LIN {X 0,Y 191.848,Z 587.295,A -85,B 0,C 180,E1 -21685.798,E2 -21685.798} C_VEL
LIN {X 0,Y 192.887,Z 588.321,A -85,B 0,C 180,E1 -21690,E2 -21690} C_VEL
LIN {X 0,Y 191.871,Z 587.279,A -85,B 0,C 180,E1 -21694.201,E2 -21694.201} C_VEL
LIN {X 0,Y 191.346,Z 585.399,A -85,B 0,C 180,E1 -21697.391,E2 -21697.391} C_VEL
LIN {X 0,Y 191.276,Z 582.566,A -85,B 0,C 180,E1 -21700.586,E2 -21700.586} C_VEL
LIN {X 0,Y 191.732,Z 578.708,A -85,B 0,C 180,E1 -21703.784,E2 -21703.784} C_VEL
LIN {X 0,Y 192.838,Z 573.752,A -85,B 0,C 180,E1 -21706.951,E2 -21706.951} C_VEL
LIN {X 0,Y 194.816,Z 567.046,A -85,B 0,C 180,E1 -21710.289,E2 -21710.289} C_VEL
LIN {X 0,Y 197.119,Z 559.922,A -85,B 0,C 180,E1 -21713.09,E2 -21713.09} C_VEL
LIN {X 0,Y 199.714,Z 552.189,A -85,B 0,C 180,E1 -21715.536,E2 -21715.536} C_VEL
LIN {X 0,Y 202.715,Z 542.86,A -85,B 0,C 180,E1 -21717.906,E2 -21717.906} C_VEL
LIN {X 0,Y 205.926,Z 532.546,A -85,B 0,C 180,E1 -21719.942,E2 -21719.942} C_VEL
LIN {X 0,Y 209.011,Z 521.131,A -85,B 0,C 180,E1 -21721.694,E2 -21721.694} C_VEL
LIN {X 0,Y 211.609,Z 509.286,A -85,B 0,C 180,E1 -21723.087,E2 -21723.087} C_VEL
LIN {X 0,Y 213.648,Z 497.038,A -85,B 0,C 180,E1 -21724.145,E2 -21724.145} C_VEL
LIN {X 0,Y 215.176,Z 483.319,A -85,B 0,C 180,E1 -21724.944,E2 -21724.944} C_VEL
LIN {X 0,Y 216.382,Z 458.003,A -85,B 0,C 180,E1 -21725.811,E2 -21725.811} C_VEL
LIN {X 0,Y 214.524,Z 429.768,A -85,B 0,C 180,E1 -21727.297,E2 -21727.297} C_VEL
LIN {X 0,Y 211.874,Z 401.366,A -85,B 0,C 180,E1 -21729.012,E2 -21729.012} C_VEL
LIN {X 0,Y 211.043,Z 395.885,A -85,B 0,C 180,E1 -21729.422,E2 -21729.422} C_VEL
LIN {X 0,Y 206.302,Z 384.53,A -85,B 0,C 180,E1 -21730.977,E2 -21730.977} C_VEL
LIN {X 0,Y 200.71,Z 373.052,A -85,B 0,C 180,E1 -21732.867,E2 -21732.867} C_VEL
LIN {X 0,Y 198.537,Z 368.397,A -85,B 0,C 180,E1 -21733.75,E2 -21733.75} C_VEL
LIN {X 0,Y 196.291,Z 359.935,A -85,B 0,C 180,E1 -21737.831,E2 -21737.831} C_VEL
LIN {X 0,Y 194.026,Z 352.255,A -85,B 0,C 180,E1 -21741.992,E2 -21741.992} C_VEL
LIN {X 0,Y 192.578,Z 347.556,A -85,B 0,C 180,E1 -21744.836,E2 -21744.836} C_VEL
LIN {X 0,Y 192.567,Z 347.483,A -85,B 0,C 180,E1 -21749.273,E2 -21749.273} C_VEL
LIN {X 0,Y 192.616,Z 347.458,A -85,B 0,C 180,E1 -21751.684,E2 -21751.684} C_VEL
LIN {X 0,Y 192.669,Z 347.47,A -85,B 0,C 180,E1 -21756.344,E2 -21756.344} C_VEL
LIN {X 0,Y 192.728,Z 347.448,A -85,B 0,C 180,E1 -21761.459,E2 -21761.459} C_VEL
LIN {X 0,Y 192.755,Z 347.462,A -85,B 0,C 180,E1 -21765.213,E2 -21765.213} C_VEL
LIN {X 0,Y 192.942,Z 347.448,A -85,B 0,C 180,E1 -21769.567,E2 -21769.567} C_VEL
LIN {X 0,Y 192.965,Z 347.423,A -85,B 0,C 180,E1 -21773.727,E2 -21773.727} C_VEL
LIN {X 0,Y 193.228,Z 347.414,A -85,B 0,C 180,E1 -21777.916,E2 -21777.916} C_VEL
LIN {X 0,Y 193.409,Z 347.368,A -85,B 0,C 180,E1 -21780,E2 -21780} C_VEL
LIN {X 0,Y 192.937,Z 347.452,A -85,B 0,C 180,E1 -21784.178,E2 -21784.178} C_VEL
LIN {X 0,Y 193.02,Z 347.415,A -85,B 0,C 180,E1 -21788.375,E2 -21788.375} C_VEL
LIN {X 0,Y 192.789,Z 347.457,A -85,B 0,C 180,E1 -21792.634,E2 -21792.634} C_VEL
LIN {X 0,Y 192.716,Z 347.474,A -85,B 0,C 180,E1 -21796.963,E2 -21796.963} C_VEL
LIN {X 0,Y 192.583,Z 347.474,A -85,B 0,C 180,E1 -21801.404,E2 -21801.404} C_VEL
LIN {X 0,Y 192.624,Z 347.491,A -85,B 0,C 180,E1 -21804.199,E2 -21804.199} C_VEL
LIN {X 0,Y 192.597,Z 347.42,A -85,B 0,C 180,E1 -21808.865,E2 -21808.865} C_VEL
LIN {X 0,Y 192.592,Z 347.466,A -85,B 0,C 180,E1 -21813.187,E2 -21813.187} C_VEL
LIN {X 0,Y 192.539,Z 347.449,A -85,B 0,C 180,E1 -21818.355,E2 -21818.355} C_VEL
LIN {X 0,Y 192.504,Z 347.505,A -85,B 0,C 180,E1 -21823.101,E2 -21823.101} C_VEL
LIN {X 0,Y 192.582,Z 347.745,A -85,B 0,C 180,E1 -21825.324,E2 -21825.324} C_VEL
LIN {X 0,Y 192.845,Z 348.9,A -85,B 0,C 180,E1 -21825.748,E2 -21825.748} C_VEL
LIN {X 0,Y 194.502,Z 351.576,A -85,B 0,C 180,E1 -21826.395,E2 -21826.395} C_VEL
LIN {X 0,Y 195.588,Z 352.693,A -85,B 0,C 180,E1 -21826.764,E2 -21826.764} C_VEL
LIN {X 0,Y 197.832,Z 356.164,A -85,B 0,C 180,E1 -21827.564,E2 -21827.564} C_VEL
LIN {X 0,Y 203.879,Z 365.281,A -85,B 0,C 180,E1 -21829.573,E2 -21829.573} C_VEL
LIN {X 0,Y 210.142,Z 375.738,A -85,B 0,C 180,E1 -21831.518,E2 -21831.518} C_VEL
LIN {X 0,Y 216.801,Z 388.352,A -85,B 0,C 180,E1 -21833.471,E2 -21833.471} C_VEL
LIN {X 0,Y 219.395,Z 393.771,A -85,B 0,C 180,E1 -21834.207,E2 -21834.207} C_VEL
LIN {X 0,Y 218.184,Z 433.029,A -85,B 0,C 180,E1 -21835.609,E2 -21835.609} C_VEL
LIN {X 0,Y 217.164,Z 446.771,A -85,B 0,C 180,E1 -21836.484,E2 -21836.484} C_VEL
LIN {X 0,Y 215.726,Z 459.041,A -85,B 0,C 180,E1 -21837.637,E2 -21837.637} C_VEL
LIN {X 0,Y 213.801,Z 470.392,A -85,B 0,C 180,E1 -21839.058,E2 -21839.058} C_VEL
LIN {X 0,Y 211.456,Z 480.568,A -85,B 0,C 180,E1 -21840.645,E2 -21840.645} C_VEL
LIN {X 0,Y 209.005,Z 489.845,A -85,B 0,C 180,E1 -21842.461,E2 -21842.461} C_VEL
LIN {X 0,Y 206.379,Z 499.292,A -85,B 0,C 180,E1 -21844.807,E2 -21844.807} C_VEL
LIN {X 0,Y 203.892,Z 507.03,A -85,B 0,C 180,E1 -21847.184,E2 -21847.184} C_VEL
LIN {X 0,Y 201.23,Z 514.686,A -85,B 0,C 180,E1 -21850.145,E2 -21850.145} C_VEL
LIN {X 0,Y 198.708,Z 521.487,A -85,B 0,C 180,E1 -21853.564,E2 -21853.564} C_VEL
LIN {X 0,Y 196.834,Z 526.095,A -85,B 0,C 180,E1 -21856.58,E2 -21856.58} C_VEL
LIN {X 0,Y 195.194,Z 529.639,A -85,B 0,C 180,E1 -21859.629,E2 -21859.629} C_VEL
LIN {X 0,Y 194.393,Z 531.461,A -85,B 0,C 180,E1 -21861.685,E2 -21861.685} C_VEL
LIN {X 0,Y 194.029,Z 532.795,A -85,B 0,C 180,E1 -21863.762,E2 -21863.762} C_VEL
LIN {X 0,Y 193.592,Z 533.767,A -85,B 0,C 180,E1 -21865.836,E2 -21865.836} C_VEL
LIN {X 0,Y 193.485,Z 534.343,A -85,B 0,C 180,E1 -21867.918,E2 -21867.918} C_VEL
LIN {X 0,Y 193.415,Z 534.565,A -85,B 0,C 180,E1 -21870,E2 -21870} C_VEL
LIN {X 0,Y 193.484,Z 534.376,A -85,B 0,C 180,E1 -21872.082,E2 -21872.082} C_VEL
LIN {X 0,Y 194.022,Z 532.87,A -85,B 0,C 180,E1 -21876.238,E2 -21876.238} C_VEL
LIN {X 0,Y 194.377,Z 531.572,A -85,B 0,C 180,E1 -21878.316,E2 -21878.316} C_VEL
LIN {X 0,Y 195.772,Z 528.732,A -85,B 0,C 180,E1 -21881.387,E2 -21881.387} C_VEL
LIN {X 0,Y 197.474,Z 524.899,A -85,B 0,C 180,E1 -21884.426,E2 -21884.426} C_VEL
LIN {X 0,Y 199.366,Z 519.811,A -85,B 0,C 180,E1 -21887.541,E2 -21887.541} C_VEL
LIN {X 0,Y 202.139,Z 512.562,A -85,B 0,C 180,E1 -21890.877,E2 -21890.877} C_VEL
LIN {X 0,Y 204.908,Z 504.527,A -85,B 0,C 180,E1 -21893.766,E2 -21893.766} C_VEL
LIN {X 0,Y 207.391,Z 496.296,A -85,B 0,C 180,E1 -21896.138,E2 -21896.138} C_VEL
LIN {X 0,Y 209.819,Z 487.254,A -85,B 0,C 180,E1 -21898.237,E2 -21898.237} C_VEL
LIN {X 0,Y 212.577,Z 476.707,A -85,B 0,C 180,E1 -21900.126,E2 -21900.126} C_VEL
LIN {X 0,Y 214.853,Z 465.168,A -85,B 0,C 180,E1 -21901.781,E2 -21901.781} C_VEL
LIN {X 0,Y 216.678,Z 453.863,A -85,B 0,C 180,E1 -21903.004,E2 -21903.004} C_VEL
LIN {X 0,Y 217.809,Z 441.291,A -85,B 0,C 180,E1 -21904.043,E2 -21904.043} C_VEL
LIN {X 0,Y 218.404,Z 428.456,A -85,B 0,C 180,E1 -21904.744,E2 -21904.744} C_VEL
LIN {X 0,Y 219.541,Z 393.957,A -85,B 0,C 180,E1 -21905.916,E2 -21905.916} C_VEL
LIN {X 0,Y 211.91,Z 378.784,A -85,B 0,C 180,E1 -21908.126,E2 -21908.126} C_VEL
LIN {X 0,Y 205.192,Z 367.34,A -85,B 0,C 180,E1 -21910.185,E2 -21910.185} C_VEL
LIN {X 0,Y 198.147,Z 356.536,A -85,B 0,C 180,E1 -21912.516,E2 -21912.516} C_VEL
LIN {X 0,Y 195.883,Z 353.302,A -85,B 0,C 180,E1 -21913.309,E2 -21913.309} C_VEL
LIN {X 0,Y 194.98,Z 352.019,A -85,B 0,C 180,E1 -21913.633,E2 -21913.633} C_VEL
LIN {X 0,Y 193.09,Z 349.489,A -85,B 0,C 180,E1 -21914.325,E2 -21914.325} C_VEL
LIN {X 0,Y 192.625,Z 347.931,A -85,B 0,C 180,E1 -21914.751,E2 -21914.751} C_VEL
LIN {X 0,Y 192.543,Z 347.583,A -85,B 0,C 180,E1 -21915.101,E2 -21915.101} C_VEL
LIN {X 0,Y 192.503,Z 347.454,A -85,B 0,C 180,E1 -21920.055,E2 -21920.055} C_VEL
LIN {X 0,Y 192.556,Z 347.486,A -85,B 0,C 180,E1 -21924.269,E2 -21924.269} C_VEL
LIN {X 0,Y 192.603,Z 347.46,A -85,B 0,C 180,E1 -21927.061,E2 -21927.061} C_VEL
LIN {X 0,Y 192.616,Z 347.421,A -85,B 0,C 180,E1 -21931.684,E2 -21931.684} C_VEL
LIN {X 0,Y 192.659,Z 347.486,A -85,B 0,C 180,E1 -21936.342,E2 -21936.342} C_VEL
LIN {X 0,Y 192.692,Z 347.48,A -85,B 0,C 180,E1 -21941.491,E2 -21941.491} C_VEL
LIN {X 0,Y 192.725,Z 347.453,A -85,B 0,C 180,E1 -21945.211,E2 -21945.211} C_VEL
LIN {X 0,Y 192.943,Z 347.447,A -85,B 0,C 180,E1 -21949.567,E2 -21949.567} C_VEL
LIN {X 0,Y 192.962,Z 347.432,A -85,B 0,C 180,E1 -21953.727,E2 -21953.727} C_VEL
LIN {X 0,Y 193.228,Z 347.394,A -85,B 0,C 180,E1 -21957.915,E2 -21957.915} C_VEL
LIN {X 0,Y 193.409,Z 347.368,A -85,B 0,C 180,E1 -21960,E2 -21960} C_VEL
LIN {X 0,Y 192.932,Z 347.439,A -85,B 0,C 180,E1 -21964.178,E2 -21964.178} C_VEL
LIN {X 0,Y 193.021,Z 347.433,A -85,B 0,C 180,E1 -21968.374,E2 -21968.374} C_VEL
LIN {X 0,Y 192.79,Z 347.445,A -85,B 0,C 180,E1 -21972.634,E2 -21972.634} C_VEL
LIN {X 0,Y 192.743,Z 347.472,A -85,B 0,C 180,E1 -21976.96,E2 -21976.96} C_VEL
LIN {X 0,Y 192.589,Z 347.45,A -85,B 0,C 180,E1 -21981.403,E2 -21981.403} C_VEL
LIN {X 0,Y 192.632,Z 347.487,A -85,B 0,C 180,E1 -21984.205,E2 -21984.205} C_VEL
LIN {X 0,Y 192.598,Z 347.461,A -85,B 0,C 180,E1 -21988.865,E2 -21988.865} C_VEL
LIN {X 0,Y 192.592,Z 347.477,A -85,B 0,C 180,E1 -21993.187,E2 -21993.187} C_VEL
LIN {X 0,Y 192.586,Z 347.766,A -85,B 0,C 180,E1 -21995.243,E2 -21995.243} C_VEL
LIN {X 0,Y 195.04,Z 355.553,A -85,B 0,C 180,E1 -21999.762,E2 -21999.762} C_VEL
LIN {X 0,Y 197.364,Z 363.876,A -85,B 0,C 180,E1 -22004.064,E2 -22004.064} C_VEL
LIN {X 0,Y 198.612,Z 368.614,A -85,B 0,C 180,E1 -22006.227,E2 -22006.227} C_VEL
LIN {X 0,Y 204.695,Z 381.021,A -85,B 0,C 180,E1 -22008.404,E2 -22008.404} C_VEL
LIN {X 0,Y 210.896,Z 395.328,A -85,B 0,C 180,E1 -22010.448,E2 -22010.448} C_VEL
LIN {X 0,Y 211.406,Z 397.261,A -85,B 0,C 180,E1 -22010.64,E2 -22010.64} C_VEL
LIN {X 0,Y 213.526,Z 416.852,A -85,B 0,C 180,E1 -22011.904,E2 -22011.904} C_VEL
LIN {X 0,Y 216.009,Z 448.818,A -85,B 0,C 180,E1 -22013.687,E2 -22013.687} C_VEL
LIN {X 0,Y 216.547,Z 458.703,A -85,B 0,C 180,E1 -22014.181,E2 -22014.181} C_VEL
LIN {X 0,Y 215.968,Z 464.541,A -85,B 0,C 180,E1 -22014.299,E2 -22014.299} C_VEL
LIN {X 0,Y 213.192,Z 474.039,A -85,B 0,C 180,E1 -22014.169,E2 -22014.169} C_VEL
LIN {X 0,Y 210.01,Z 483.484,A -85,B 0,C 180,E1 -22014.056,E2 -22014.056} C_VEL
LIN {X 0,Y 208.832,Z 489.253,A -85,B 0,C 180,E1 -22014.263,E2 -22014.263} C_VEL
LIN {X 0,Y 207.17,Z 500.744,A -85,B 0,C 180,E1 -22015.078,E2 -22015.078} C_VEL
LIN {X 0,Y 205.007,Z 511.757,A -85,B 0,C 180,E1 -22016.147,E2 -22016.147} C_VEL
LIN {X 0,Y 202.148,Z 523.63,A -85,B 0,C 180,E1 -22017.688,E2 -22017.688} C_VEL
LIN {X 0,Y 198.624,Z 535.483,A -85,B 0,C 180,E1 -22019.721,E2 -22019.721} C_VEL
LIN {X 0,Y 195.149,Z 546.05,A -85,B 0,C 180,E1 -22022.085,E2 -22022.085} C_VEL
LIN {X 0,Y 192.136,Z 554.643,A -85,B 0,C 180,E1 -22024.546,E2 -22024.546} C_VEL
LIN {X 0,Y 189.191,Z 563.086,A -85,B 0,C 180,E1 -22027.619,E2 -22027.619} C_VEL
LIN {X 0,Y 186.75,Z 569.919,A -85,B 0,C 180,E1 -22030.775,E2 -22030.775} C_VEL
LIN {X 0,Y 185.118,Z 576.286,A -85,B 0,C 180,E1 -22034.588,E2 -22034.588} C_VEL
LIN {X 0,Y 184.32,Z 580.472,A -85,B 0,C 180,E1 -22037.895,E2 -22037.895} C_VEL
LIN {X 0,Y 184.177,Z 583.631,A -85,B 0,C 180,E1 -22041.22,E2 -22041.22} C_VEL
LIN {X 0,Y 184.38,Z 585.174,A -85,B 0,C 180,E1 -22043.434,E2 -22043.434} C_VEL
LIN {X 0,Y 184.755,Z 586.306,A -85,B 0,C 180,E1 -22045.637,E2 -22045.637} C_VEL
LIN {X 0,Y 185.837,Z 587.34,A -85,B 0,C 180,E1 -22050,E2 -22050} C_VEL
LIN {X 0,Y 184.774,Z 586.288,A -85,B 0,C 180,E1 -22054.363,E2 -22054.363} C_VEL
LIN {X 0,Y 184.289,Z 584.561,A -85,B 0,C 180,E1 -22057.461,E2 -22057.461} C_VEL
LIN {X 0,Y 184.232,Z 581.567,A -85,B 0,C 180,E1 -22060.996,E2 -22060.996} C_VEL
LIN {X 0,Y 184.764,Z 577.708,A -85,B 0,C 180,E1 -22064.314,E2 -22064.314} C_VEL
LIN {X 0,Y 185.968,Z 572.749,A -85,B 0,C 180,E1 -22067.597,E2 -22067.597} C_VEL
LIN {X 0,Y 187.904,Z 566.664,A -85,B 0,C 180,E1 -22070.763,E2 -22070.763} C_VEL
LIN {X 0,Y 190.556,Z 558.924,A -85,B 0,C 180,E1 -22073.934,E2 -22073.934} C_VEL
LIN {X 0,Y 193.301,Z 551.194,A -85,B 0,C 180,E1 -22076.447,E2 -22076.447} C_VEL
LIN {X 0,Y 196.459,Z 541.868,A -85,B 0,C 180,E1 -22078.877,E2 -22078.877} C_VEL
LIN {X 0,Y 199.812,Z 531.555,A -85,B 0,C 180,E1 -22080.957,E2 -22080.957} C_VEL
LIN {X 0,Y 203.013,Z 520.14,A -85,B 0,C 180,E1 -22082.745,E2 -22082.745} C_VEL
LIN {X 0,Y 205.657,Z 508.286,A -85,B 0,C 180,E1 -22084.174,E2 -22084.174} C_VEL
LIN {X 0,Y 207.798,Z 496.149,A -85,B 0,C 180,E1 -22085.236,E2 -22085.236} C_VEL
LIN {X 0,Y 209.337,Z 482.771,A -85,B 0,C 180,E1 -22086.039,E2 -22086.039} C_VEL
LIN {X 0,Y 210.605,Z 459.13,A -85,B 0,C 180,E1 -22086.864,E2 -22086.864} C_VEL
LIN {X 0,Y 208.769,Z 429.728,A -85,B 0,C 180,E1 -22088.468,E2 -22088.468} C_VEL
LIN {X 0,Y 205.982,Z 399.581,A -85,B 0,C 180,E1 -22090.383,E2 -22090.383} C_VEL
LIN {X 0,Y 202.843,Z 391.689,A -85,B 0,C 180,E1 -22091.474,E2 -22091.474} C_VEL
LIN {X 0,Y 196.692,Z 378.218,A -85,B 0,C 180,E1 -22093.673,E2 -22093.673} C_VEL
LIN {X 0,Y 193.129,Z 371.46,A -85,B 0,C 180,E1 -22094.996,E2 -22094.996} C_VEL
LIN {X 0,Y 190.941,Z 366.871,A -85,B 0,C 180,E1 -22095.994,E2 -22095.994} C_VEL
LIN {X 0,Y 188.512,Z 358.02,A -85,B 0,C 180,E1 -22100.67,E2 -22100.67} C_VEL
LIN {X 0,Y 186.002,Z 350.11,A -85,B 0,C 180,E1 -22105.475,E2 -22105.475} C_VEL
LIN {X 0,Y 185.573,Z 348.398,A -85,B 0,C 180,E1 -22106.64,E2 -22106.64} C_VEL
LIN {X 0,Y 185.544,Z 348.342,A -85,B 0,C 180,E1 -22110.595,E2 -22110.595} C_VEL
LIN {X 0,Y 185.578,Z 348.369,A -85,B 0,C 180,E1 -22115.381,E2 -22115.381} C_VEL
LIN {X 0,Y 185.67,Z 348.321,A -85,B 0,C 180,E1 -22121.135,E2 -22121.135} C_VEL
LIN {X 0,Y 185.687,Z 348.35,A -85,B 0,C 180,E1 -22124.637,E2 -22124.637} C_VEL
LIN {X 0,Y 185.885,Z 348.325,A -85,B 0,C 180,E1 -22129.419,E2 -22129.419} C_VEL
LIN {X 0,Y 185.93,Z 348.299,A -85,B 0,C 180,E1 -22133.489,E2 -22133.489} C_VEL
LIN {X 0,Y 186.173,Z 348.293,A -85,B 0,C 180,E1 -22137.837,E2 -22137.837} C_VEL
LIN {X 0,Y 186.375,Z 348.244,A -85,B 0,C 180,E1 -22140,E2 -22140} C_VEL
LIN {X 0,Y 185.885,Z 348.33,A -85,B 0,C 180,E1 -22144.337,E2 -22144.337} C_VEL
LIN {X 0,Y 185.97,Z 348.295,A -85,B 0,C 180,E1 -22148.695,E2 -22148.695} C_VEL
LIN {X 0,Y 185.714,Z 348.332,A -85,B 0,C 180,E1 -22153.124,E2 -22153.124} C_VEL
LIN {X 0,Y 185.653,Z 348.359,A -85,B 0,C 180,E1 -22157.629,E2 -22157.629} C_VEL
LIN {X 0,Y 185.55,Z 348.355,A -85,B 0,C 180,E1 -22162.257,E2 -22162.257} C_VEL
LIN {X 0,Y 185.497,Z 348.324,A -85,B 0,C 180,E1 -22167.043,E2 -22167.043} C_VEL
LIN {X 0,Y 185.541,Z 348.296,A -85,B 0,C 180,E1 -22169.5,E2 -22169.5} C_VEL
LIN {X 0,Y 185.495,Z 348.38,A -85,B 0,C 180,E1 -22174.633,E2 -22174.633} C_VEL
LIN {X 0,Y 185.498,Z 348.335,A -85,B 0,C 180,E1 -22177.315,E2 -22177.315} C_VEL
LIN {X 0,Y 185.49,Z 348.481,A -85,B 0,C 180,E1 -22182.922,E2 -22182.922} C_VEL
LIN {X 0,Y 185.708,Z 349.527,A -85,B 0,C 180,E1 -22183.499,E2 -22183.499} C_VEL
LIN {X 0,Y 187.062,Z 352.077,A -85,B 0,C 180,E1 -22184.129,E2 -22184.129} C_VEL
LIN {X 0,Y 188.825,Z 353.884,A -85,B 0,C 180,E1 -22184.794,E2 -22184.794} C_VEL
LIN {X 0,Y 191.08,Z 357.305,A -85,B 0,C 180,E1 -22185.675,E2 -22185.675} C_VEL
LIN {X 0,Y 195.742,Z 364.087,A -85,B 0,C 180,E1 -22187.376,E2 -22187.376} C_VEL
LIN {X 0,Y 202.922,Z 375.487,A -85,B 0,C 180,E1 -22189.806,E2 -22189.806} C_VEL
LIN {X 0,Y 209.873,Z 388.222,A -85,B 0,C 180,E1 -22191.998,E2 -22191.998} C_VEL
LIN {X 0,Y 213.666,Z 396.039,A -85,B 0,C 180,E1 -22193.144,E2 -22193.144} C_VEL
LIN {X 0,Y 212.389,Z 434.304,A -85,B 0,C 180,E1 -22194.549,E2 -22194.549} C_VEL
LIN {X 0,Y 211.33,Z 447.834,A -85,B 0,C 180,E1 -22195.437,E2 -22195.437} C_VEL
LIN {X 0,Y 209.822,Z 460.026,A -85,B 0,C 180,E1 -22196.61,E2 -22196.61} C_VEL
LIN {X 0,Y 207.841,Z 471.183,A -85,B 0,C 180,E1 -22198.032,E2 -22198.032} C_VEL
LIN {X 0,Y 205.359,Z 481.55,A -85,B 0,C 180,E1 -22199.683,E2 -22199.683} C_VEL
LIN {X 0,Y 202.797,Z 490.827,A -85,B 0,C 180,E1 -22201.543,E2 -22201.543} C_VEL
LIN {X 0,Y 200.041,Z 500.273,A -85,B 0,C 180,E1 -22203.95,E2 -22203.95} C_VEL
LIN {X 0,Y 197.433,Z 508.01,A -85,B 0,C 180,E1 -22206.393,E2 -22206.393} C_VEL
LIN {X 0,Y 194.634,Z 515.666,A -85,B 0,C 180,E1 -22209.442,E2 -22209.442} C_VEL
LIN {X 0,Y 191.978,Z 522.466,A -85,B 0,C 180,E1 -22212.971,E2 -22212.971} C_VEL
LIN {X 0,Y 190.005,Z 527.074,A -85,B 0,C 180,E1 -22216.089,E2 -22216.089} C_VEL
LIN {X 0,Y 188.282,Z 530.618,A -85,B 0,C 180,E1 -22219.244,E2 -22219.244} C_VEL
LIN {X 0,Y 187.438,Z 532.441,A -85,B 0,C 180,E1 -22221.374,E2 -22221.374} C_VEL
LIN {X 0,Y 187.042,Z 533.773,A -85,B 0,C 180,E1 -22223.528,E2 -22223.528} C_VEL
LIN {X 0,Y 186.583,Z 534.745,A -85,B 0,C 180,E1 -22225.68,E2 -22225.68} C_VEL
LIN {X 0,Y 186.462,Z 535.321,A -85,B 0,C 180,E1 -22227.84,E2 -22227.84} C_VEL
LIN {X 0,Y 186.388,Z 535.543,A -85,B 0,C 180,E1 -22230,E2 -22230} C_VEL
LIN {X 0,Y 186.461,Z 535.354,A -85,B 0,C 180,E1 -22232.16,E2 -22232.16} C_VEL
LIN {X 0,Y 187.035,Z 533.848,A -85,B 0,C 180,E1 -22236.472,E2 -22236.472} C_VEL
LIN {X 0,Y 187.421,Z 532.55,A -85,B 0,C 180,E1 -22238.626,E2 -22238.626} C_VEL
LIN {X 0,Y 188.888,Z 529.71,A -85,B 0,C 180,E1 -22241.808,E2 -22241.808} C_VEL
LIN {X 0,Y 190.676,Z 525.876,A -85,B 0,C 180,E1 -22244.952,E2 -22244.952} C_VEL
LIN {X 0,Y 192.676,Z 520.788,A -85,B 0,C 180,E1 -22248.171,E2 -22248.171} C_VEL
LIN {X 0,Y 195.588,Z 513.538,A -85,B 0,C 180,E1 -22251.611,E2 -22251.611} C_VEL
LIN {X 0,Y 198.496,Z 505.503,A -85,B 0,C 180,E1 -22254.583,E2 -22254.583} C_VEL
LIN {X 0,Y 201.103,Z 497.272,A -85,B 0,C 180,E1 -22257.02,E2 -22257.02} C_VEL
LIN {X 0,Y 203.66,Z 488.227,A -85,B 0,C 180,E1 -22259.171,E2 -22259.171} C_VEL
LIN {X 0,Y 206.799,Z 476.655,A -85,B 0,C 180,E1 -22261.266,E2 -22261.266} C_VEL
LIN {X 0,Y 209.196,Z 464.702,A -85,B 0,C 180,E1 -22262.978,E2 -22262.978} C_VEL
LIN {X 0,Y 211.103,Z 452.077,A -85,B 0,C 180,E1 -22264.309,E2 -22264.309} C_VEL
LIN {X 0,Y 212.274,Z 439.226,A -85,B 0,C 180,E1 -22265.301,E2 -22265.301} C_VEL
LIN {X 0,Y 212.795,Z 425.544,A -85,B 0,C 180,E1 -22265.973,E2 -22265.973} C_VEL
LIN {X 0,Y 213.782,Z 396.205,A -85,B 0,C 180,E1 -22266.989,E2 -22266.989} C_VEL
LIN {X 0,Y 206.699,Z 382.077,A -85,B 0,C 180,E1 -22269.162,E2 -22269.162} C_VEL
LIN {X 0,Y 200.469,Z 371.475,A -85,B 0,C 180,E1 -22271.179,E2 -22271.179} C_VEL
LIN {X 0,Y 194.162,Z 361.696,A -85,B 0,C 180,E1 -22273.379,E2 -22273.379} C_VEL
LIN {X 0,Y 191.048,Z 357.25,A -85,B 0,C 180,E1 -22274.532,E2 -22274.532} C_VEL
LIN {X 0,Y 188.907,Z 354.019,A -85,B 0,C 180,E1 -22275.37,E2 -22275.37} C_VEL
LIN {X 0,Y 186.163,Z 350.725,A -85,B 0,C 180,E1 -22276.446,E2 -22276.446} C_VEL
LIN {X 0,Y 185.603,Z 349.075,A -85,B 0,C 180,E1 -22276.845,E2 -22276.845} C_VEL
LIN {X 0,Y 185.444,Z 348.432,A -85,B 0,C 180,E1 -22277.457,E2 -22277.457} C_VEL
LIN {X 0,Y 185.499,Z 348.334,A -85,B 0,C 180,E1 -22282.713,E2 -22282.713} C_VEL
LIN {X 0,Y 185.528,Z 348.319,A -85,B 0,C 180,E1 -22287.972,E2 -22287.972} C_VEL
LIN {X 0,Y 185.545,Z 348.296,A -85,B 0,C 180,E1 -22290.595,E2 -22290.595} C_VEL
LIN {X 0,Y 185.56,Z 348.368,A -85,B 0,C 180,E1 -22295.378,E2 -22295.378} C_VEL
LIN {X 0,Y 185.622,Z 348.356,A -85,B 0,C 180,E1 -22301.178,E2 -22301.178} C_VEL
LIN {X 0,Y 185.656,Z 348.335,A -85,B 0,C 180,E1 -22304.634,E2 -22304.634} C_VEL
LIN {X 0,Y 185.885,Z 348.327,A -85,B 0,C 180,E1 -22309.419,E2 -22309.419} C_VEL
LIN {X 0,Y 185.927,Z 348.305,A -85,B 0,C 180,E1 -22313.489,E2 -22313.489} C_VEL
LIN {X 0,Y 186.174,Z 348.273,A -85,B 0,C 180,E1 -22317.836,E2 -22317.836} C_VEL
LIN {X 0,Y 186.375,Z 348.244,A -85,B 0,C 180,E1 -22320,E2 -22320} C_VEL
LIN {X 0,Y 185.88,Z 348.314,A -85,B 0,C 180,E1 -22324.337,E2 -22324.337} C_VEL
LIN {X 0,Y 185.971,Z 348.314,A -85,B 0,C 180,E1 -22328.694,E2 -22328.694} C_VEL
LIN {X 0,Y 185.717,Z 348.326,A -85,B 0,C 180,E1 -22333.124,E2 -22333.124} C_VEL
LIN {X 0,Y 185.68,Z 348.339,A -85,B 0,C 180,E1 -22337.626,E2 -22337.626} C_VEL
LIN {X 0,Y 185.556,Z 348.333,A -85,B 0,C 180,E1 -22342.256,E2 -22342.256} C_VEL
LIN {X 0,Y 185.575,Z 348.37,A -85,B 0,C 180,E1 -22344.646,E2 -22344.646} C_VEL
LIN {X 0,Y 185.541,Z 348.343,A -85,B 0,C 180,E1 -22349.5,E2 -22349.5} C_VEL
LIN {X 0,Y 185.574,Z 348.537,A -85,B 0,C 180,E1 -22353.36,E2 -22353.36} C_VEL
LIN {X 0,Y 187.999,Z 356.388,A -85,B 0,C 180,E1 -22358.276,E2 -22358.276} C_VEL
LIN {X 0,Y 190.101,Z 363.648,A -85,B 0,C 180,E1 -22362.321,E2 -22362.321} C_VEL
LIN {X 0,Y 191.108,Z 367.307,A -85,B 0,C 180,E1 -22364.049,E2 -22364.049} C_VEL
LIN {X 0,Y 197.324,Z 379.464,A -85,B 0,C 180,E1 -22366.465,E2 -22366.465} C_VEL
LIN {X 0,Y 202.276,Z 390.248,A -85,B 0,C 180,E1 -22368.238,E2 -22368.238} C_VEL
LIN {X 0,Y 205.96,Z 399.37,A -85,B 0,C 180,E1 -22369.522,E2 -22369.522} C_VEL
LIN {X 0,Y 207.784,Z 416.829,A -85,B 0,C 180,E1 -22370.694,E2 -22370.694} C_VEL
LIN {X 0,Y 210.117,Z 447.801,A -85,B 0,C 180,E1 -22372.497,E2 -22372.497} C_VEL
LIN {X 0,Y 210.729,Z 459.603,A -85,B 0,C 180,E1 -22373.108,E2 -22373.108} C_VEL
LIN {X 0,Y 209.472,Z 482.581,A -85,B 0,C 180,E1 -22373.904,E2 -22373.904} C_VEL
LIN {X 0,Y 208.832,Z 489.253,A -85,B 0,C 180,E1 -22374.263,E2 -22374.263} C_VEL
LIN {X 0,Y 207.517,Z 494.952,A -85,B 0,C 180,E1 -22374.523,E2 -22374.523} C_VEL
LIN {X 0,Y 203.565,Z 504.016,A -85,B 0,C 180,E1 -22374.819,E2 -22374.819} C_VEL
LIN {X 0,Y 199.256,Z 512.783,A -85,B 0,C 180,E1 -22375.322,E2 -22375.322} C_VEL
LIN {X 0,Y 197.399,Z 518.01,A -85,B 0,C 180,E1 -22375.911,E2 -22375.911} C_VEL
LIN {X 0,Y 194.137,Z 529.566,A -85,B 0,C 180,E1 -22377.727,E2 -22377.727} C_VEL
LIN {X 0,Y 190.664,Z 540.069,A -85,B 0,C 180,E1 -22379.853,E2 -22379.853} C_VEL
LIN {X 0,Y 187.57,Z 548.69,A -85,B 0,C 180,E1 -22382.073,E2 -22382.073} C_VEL
LIN {X 0,Y 184.586,Z 556.683,A -85,B 0,C 180,E1 -22384.638,E2 -22384.638} C_VEL
LIN {X 0,Y 181.693,Z 564.669,A -85,B 0,C 180,E1 -22387.905,E2 -22387.905} C_VEL
LIN {X 0,Y 179.676,Z 569.955,A -85,B 0,C 180,E1 -22390.581,E2 -22390.581} C_VEL
LIN {X 0,Y 178.223,Z 575.29,A -85,B 0,C 180,E1 -22393.976,E2 -22393.976} C_VEL
LIN {X 0,Y 177.327,Z 579.477,A -85,B 0,C 180,E1 -22397.41,E2 -22397.41} C_VEL
LIN {X 0,Y 177.117,Z 582.637,A -85,B 0,C 180,E1 -22400.868,E2 -22400.868} C_VEL
LIN {X 0,Y 177.298,Z 584.182,A -85,B 0,C 180,E1 -22403.17,E2 -22403.17} C_VEL
LIN {X 0,Y 177.665,Z 585.316,A -85,B 0,C 180,E1 -22405.462,E2 -22405.462} C_VEL
LIN {X 0,Y 178.757,Z 586.355,A -85,B 0,C 180,E1 -22410,E2 -22410} C_VEL
LIN {X 0,Y 177.68,Z 585.298,A -85,B 0,C 180,E1 -22414.537,E2 -22414.537} C_VEL
LIN {X 0,Y 177.215,Z 583.749,A -85,B 0,C 180,E1 -22417.498,E2 -22417.498} C_VEL
LIN {X 0,Y 177.18,Z 580.566,A -85,B 0,C 180,E1 -22421.439,E2 -22421.439} C_VEL
LIN {X 0,Y 177.828,Z 576.709,A -85,B 0,C 180,E1 -22424.885,E2 -22424.885} C_VEL
LIN {X 0,Y 179.126,Z 571.747,A -85,B 0,C 180,E1 -22428.293,E2 -22428.293} C_VEL
LIN {X 0,Y 181.039,Z 566.224,A -85,B 0,C 180,E1 -22431.3,E2 -22431.3} C_VEL
LIN {X 0,Y 184.038,Z 557.927,A -85,B 0,C 180,E1 -22434.838,E2 -22434.838} C_VEL
LIN {X 0,Y 186.947,Z 550.2,A -85,B 0,C 180,E1 -22437.42,E2 -22437.42} C_VEL
LIN {X 0,Y 190.274,Z 540.877,A -85,B 0,C 180,E1 -22439.909,E2 -22439.909} C_VEL
LIN {X 0,Y 193.771,Z 530.565,A -85,B 0,C 180,E1 -22442.035,E2 -22442.035} C_VEL
LIN {X 0,Y 197.081,Z 519.147,A -85,B 0,C 180,E1 -22443.861,E2 -22443.861} C_VEL
LIN {X 0,Y 199.768,Z 507.282,A -85,B 0,C 180,E1 -22445.329,E2 -22445.329} C_VEL
LIN {X 0,Y 202.135,Z 494.591,A -85,B 0,C 180,E1 -22446.435,E2 -22446.435} C_VEL
LIN {X 0,Y 203.702,Z 481.124,A -85,B 0,C 180,E1 -22447.245,E2 -22447.245} C_VEL
LIN {X 0,Y 204.811,Z 459.197,A -85,B 0,C 180,E1 -22448.042,E2 -22448.042} C_VEL
LIN {X 0,Y 203.182,Z 431.115,A -85,B 0,C 180,E1 -22449.624,E2 -22449.624} C_VEL
LIN {X 0,Y 200.661,Z 402.075,A -85,B 0,C 180,E1 -22451.527,E2 -22451.527} C_VEL
LIN {X 0,Y 196.572,Z 392.063,A -85,B 0,C 180,E1 -22453.035,E2 -22453.035} C_VEL
LIN {X 0,Y 191.359,Z 380.954,A -85,B 0,C 180,E1 -22455.023,E2 -22455.023} C_VEL
LIN {X 0,Y 188.706,Z 375.764,A -85,B 0,C 180,E1 -22456.08,E2 -22456.08} C_VEL
LIN {X 0,Y 185.981,Z 370.594,A -85,B 0,C 180,E1 -22457.21,E2 -22457.21} C_VEL
LIN {X 0,Y 183.329,Z 365.354,A -85,B 0,C 180,E1 -22458.51,E2 -22458.51} C_VEL
LIN {X 0,Y 181.403,Z 358.559,A -85,B 0,C 180,E1 -22462.396,E2 -22462.396} C_VEL
LIN {X 0,Y 179.348,Z 351.874,A -85,B 0,C 180,E1 -22466.728,E2 -22466.728} C_VEL
LIN {X 0,Y 178.46,Z 349.277,A -85,B 0,C 180,E1 -22468.712,E2 -22468.712} C_VEL
LIN {X 0,Y 178.482,Z 349.244,A -85,B 0,C 180,E1 -22474.333,E2 -22474.333} C_VEL
LIN {X 0,Y 178.512,Z 349.2,A -85,B 0,C 180,E1 -22479.248,E2 -22479.248} C_VEL
LIN {X 0,Y 178.645,Z 349.202,A -85,B 0,C 180,E1 -22481.656,E2 -22481.656} C_VEL
LIN {X 0,Y 178.651,Z 349.208,A -85,B 0,C 180,E1 -22486.347,E2 -22486.347} C_VEL
LIN {X 0,Y 178.903,Z 349.198,A -85,B 0,C 180,E1 -22490.959,E2 -22490.959} C_VEL
LIN {X 0,Y 179.121,Z 349.172,A -85,B 0,C 180,E1 -22497.751,E2 -22497.751} C_VEL
LIN {X 0,Y 179.341,Z 349.12,A -85,B 0,C 180,E1 -22500,E2 -22500} C_VEL
LIN {X 0,Y 178.834,Z 349.208,A -85,B 0,C 180,E1 -22504.508,E2 -22504.508} C_VEL
LIN {X 0,Y 178.901,Z 349.177,A -85,B 0,C 180,E1 -22509.041,E2 -22509.041} C_VEL
LIN {X 0,Y 178.641,Z 349.208,A -85,B 0,C 180,E1 -22513.654,E2 -22513.654} C_VEL
LIN {X 0,Y 178.554,Z 349.231,A -85,B 0,C 180,E1 -22519.154,E2 -22519.154} C_VEL
LIN {X 0,Y 178.502,Z 349.238,A -85,B 0,C 180,E1 -22525.104,E2 -22525.104} C_VEL
LIN {X 0,Y 178.458,Z 349.182,A -85,B 0,C 180,E1 -22530.795,E2 -22530.795} C_VEL
LIN {X 0,Y 178.48,Z 349.246,A -85,B 0,C 180,E1 -22534.219,E2 -22534.219} C_VEL
LIN {X 0,Y 178.439,Z 349.308,A -85,B 0,C 180,E1 -22540.254,E2 -22540.254} C_VEL
LIN {X 0,Y 178.591,Z 350.157,A -85,B 0,C 180,E1 -22540.948,E2 -22540.948} C_VEL
LIN {X 0,Y 180.073,Z 352.989,A -85,B 0,C 180,E1 -22541.754,E2 -22541.754} C_VEL
LIN {X 0,Y 181.926,Z 354.859,A -85,B 0,C 180,E1 -22542.536,E2 -22542.536} C_VEL
LIN {X 0,Y 183.989,Z 358.073,A -85,B 0,C 180,E1 -22543.438,E2 -22543.438} C_VEL
LIN {X 0,Y 185.339,Z 359.747,A -85,B 0,C 180,E1 -22543.986,E2 -22543.986} C_VEL
LIN {X 0,Y 191.733,Z 369.148,A -85,B 0,C 180,E1 -22546.484,E2 -22546.484} C_VEL
LIN {X 0,Y 198.179,Z 379.519,A -85,B 0,C 180,E1 -22548.788,E2 -22548.788} C_VEL
LIN {X 0,Y 205.172,Z 392.498,A -85,B 0,C 180,E1 -22551.118,E2 -22551.118} C_VEL
LIN {X 0,Y 207.957,Z 398.303,A -85,B 0,C 180,E1 -22552.01,E2 -22552.01} C_VEL
LIN {X 0,Y 206.743,Z 434.634,A -85,B 0,C 180,E1 -22553.383,E2 -22553.383} C_VEL
LIN {X 0,Y 205.648,Z 448.224,A -85,B 0,C 180,E1 -22554.28,E2 -22554.28} C_VEL
LIN {X 0,Y 203.989,Z 461.011,A -85,B 0,C 180,E1 -22555.523,E2 -22555.523} C_VEL
LIN {X 0,Y 201.672,Z 473.336,A -85,B 0,C 180,E1 -22557.155,E2 -22557.155} C_VEL
LIN {X 0,Y 198.99,Z 483.803,A -85,B 0,C 180,E1 -22558.901,E2 -22558.901} C_VEL
LIN {X 0,Y 196.369,Z 492.853,A -85,B 0,C 180,E1 -22560.815,E2 -22560.815} C_VEL
LIN {X 0,Y 193.75,Z 501.254,A -85,B 0,C 180,E1 -22563.037,E2 -22563.037} C_VEL
LIN {X 0,Y 191.013,Z 508.99,A -85,B 0,C 180,E1 -22565.549,E2 -22565.549} C_VEL
LIN {X 0,Y 188.07,Z 516.646,A -85,B 0,C 180,E1 -22568.69,E2 -22568.69} C_VEL
LIN {X 0,Y 185.269,Z 523.446,A -85,B 0,C 180,E1 -22572.334,E2 -22572.334} C_VEL
LIN {X 0,Y 183.191,Z 528.053,A -85,B 0,C 180,E1 -22575.56,E2 -22575.56} C_VEL
LIN {X 0,Y 181.379,Z 531.598,A -85,B 0,C 180,E1 -22578.829,E2 -22578.829} C_VEL
LIN {X 0,Y 180.489,Z 533.42,A -85,B 0,C 180,E1 -22581.04,E2 -22581.04} C_VEL
LIN {X 0,Y 180.059,Z 534.752,A -85,B 0,C 180,E1 -22583.276,E2 -22583.276} C_VEL
LIN {X 0,Y 179.575,Z 535.724,A -85,B 0,C 180,E1 -22585.511,E2 -22585.511} C_VEL
LIN {X 0,Y 179.439,Z 536.299,A -85,B 0,C 180,E1 -22587.755,E2 -22587.755} C_VEL
LIN {X 0,Y 179.36,Z 536.521,A -85,B 0,C 180,E1 -22590,E2 -22590} C_VEL
LIN {X 0,Y 179.438,Z 536.331,A -85,B 0,C 180,E1 -22592.245,E2 -22592.245} C_VEL
LIN {X 0,Y 180.052,Z 534.826,A -85,B 0,C 180,E1 -22596.725,E2 -22596.725} C_VEL
LIN {X 0,Y 180.472,Z 533.528,A -85,B 0,C 180,E1 -22598.961,E2 -22598.961} C_VEL
LIN {X 0,Y 182.014,Z 530.687,A -85,B 0,C 180,E1 -22602.261,E2 -22602.261} C_VEL
LIN {X 0,Y 183.894,Z 526.853,A -85,B 0,C 180,E1 -22605.517,E2 -22605.517} C_VEL
LIN {X 0,Y 186.012,Z 521.764,A -85,B 0,C 180,E1 -22608.846,E2 -22608.846} C_VEL
LIN {X 0,Y 189.072,Z 514.514,A -85,B 0,C 180,E1 -22612.395,E2 -22612.395} C_VEL
LIN {X 0,Y 192.126,Z 506.478,A -85,B 0,C 180,E1 -22615.455,E2 -22615.455} C_VEL
LIN {X 0,Y 194.867,Z 498.247,A -85,B 0,C 180,E1 -22617.959,E2 -22617.959} C_VEL
LIN {X 0,Y 197.546,Z 489.202,A -85,B 0,C 180,E1 -22620.166,E2 -22620.166} C_VEL
LIN {X 0,Y 200.822,Z 477.631,A -85,B 0,C 180,E1 -22622.306,E2 -22622.306} C_VEL
LIN {X 0,Y 203.336,Z 465.674,A -85,B 0,C 180,E1 -22624.056,E2 -22624.056} C_VEL
LIN {X 0,Y 205.334,Z 453.046,A -85,B 0,C 180,E1 -22625.415,E2 -22625.415} C_VEL
LIN {X 0,Y 206.558,Z 440.471,A -85,B 0,C 180,E1 -22626.409,E2 -22626.409} C_VEL
LIN {X 0,Y 207.097,Z 427.301,A -85,B 0,C 180,E1 -22627.092,E2 -22627.092} C_VEL
LIN {X 0,Y 208.11,Z 398.489,A -85,B 0,C 180,E1 -22628.117,E2 -22628.117} C_VEL
LIN {X 0,Y 201.059,Z 384.539,A -85,B 0,C 180,E1 -22630.415,E2 -22630.415} C_VEL
LIN {X 0,Y 194.31,Z 373.108,A -85,B 0,C 180,E1 -22632.762,E2 -22632.762} C_VEL
LIN {X 0,Y 189.465,Z 365.801,A -85,B 0,C 180,E1 -22634.566,E2 -22634.566} C_VEL
LIN {X 0,Y 186.95,Z 362.139,A -85,B 0,C 180,E1 -22635.557,E2 -22635.557} C_VEL
LIN {X 0,Y 184.42,Z 358.542,A -85,B 0,C 180,E1 -22636.594,E2 -22636.594} C_VEL
LIN {X 0,Y 182.078,Z 355.187,A -85,B 0,C 180,E1 -22637.602,E2 -22637.602} C_VEL
LIN {X 0,Y 181.303,Z 354.147,A -85,B 0,C 180,E1 -22637.941,E2 -22637.941} C_VEL
LIN {X 0,Y 179.202,Z 351.718,A -85,B 0,C 180,E1 -22638.865,E2 -22638.865} C_VEL
LIN {X 0,Y 178.539,Z 349.871,A -85,B 0,C 180,E1 -22639.394,E2 -22639.394} C_VEL
LIN {X 0,Y 178.398,Z 349.267,A -85,B 0,C 180,E1 -22640.195,E2 -22640.195} C_VEL
LIN {X 0,Y 178.481,Z 349.248,A -85,B 0,C 180,E1 -22645.781,E2 -22645.781} C_VEL
LIN {X 0,Y 178.479,Z 349.175,A -85,B 0,C 180,E1 -22650.03,E2 -22650.03} C_VEL
LIN {X 0,Y 178.502,Z 349.237,A -85,B 0,C 180,E1 -22654.896,E2 -22654.896} C_VEL
LIN {X 0,Y 178.604,Z 349.236,A -85,B 0,C 180,E1 -22661.651,E2 -22661.651} C_VEL
LIN {X 0,Y 178.635,Z 349.21,A -85,B 0,C 180,E1 -22666.346,E2 -22666.346} C_VEL
LIN {X 0,Y 178.901,Z 349.178,A -85,B 0,C 180,E1 -22670.959,E2 -22670.959} C_VEL
LIN {X 0,Y 179.121,Z 349.151,A -85,B 0,C 180,E1 -22677.751,E2 -22677.751} C_VEL
LIN {X 0,Y 179.34,Z 349.119,A -85,B 0,C 180,E1 -22680,E2 -22680} C_VEL
LIN {X 0,Y 178.829,Z 349.19,A -85,B 0,C 180,E1 -22684.508,E2 -22684.508} C_VEL
LIN {X 0,Y 178.902,Z 349.198,A -85,B 0,C 180,E1 -22689.041,E2 -22689.041} C_VEL
LIN {X 0,Y 178.646,Z 349.209,A -85,B 0,C 180,E1 -22693.653,E2 -22693.653} C_VEL
LIN {X 0,Y 178.605,Z 349.195,A -85,B 0,C 180,E1 -22699.201,E2 -22699.201} C_VEL
LIN {X 0,Y 178.513,Z 349.248,A -85,B 0,C 180,E1 -22705.111,E2 -22705.111} C_VEL
LIN {X 0,Y 178.458,Z 349.251,A -85,B 0,C 180,E1 -22710.795,E2 -22710.795} C_VEL
LIN {X 0,Y 178.506,Z 349.528,A -85,B 0,C 180,E1 -22711.444,E2 -22711.444} C_VEL
LIN {X 0,Y 180.506,Z 355.774,A -85,B 0,C 180,E1 -22715.734,E2 -22715.734} C_VEL
LIN {X 0,Y 182.713,Z 363.066,A -85,B 0,C 180,E1 -22720.178,E2 -22720.178} C_VEL
LIN {X 0,Y 183.507,Z 365.742,A -85,B 0,C 180,E1 -22721.532,E2 -22721.532} C_VEL
LIN {X 0,Y 186.508,Z 371.371,A -85,B 0,C 180,E1 -22722.893,E2 -22722.893} C_VEL
LIN {X 0,Y 192.779,Z 383.64,A -85,B 0,C 180,E1 -22725.422,E2 -22725.422} C_VEL
LIN {X 0,Y 197.753,Z 394.745,A -85,B 0,C 180,E1 -22727.312,E2 -22727.312} C_VEL
LIN {X 0,Y 200.663,Z 402.019,A -85,B 0,C 180,E1 -22728.386,E2 -22728.386} C_VEL
LIN {X 0,Y 202.458,Z 420.284,A -85,B 0,C 180,E1 -22729.647,E2 -22729.647} C_VEL
LIN {X 0,Y 204.615,Z 451.483,A -85,B 0,C 180,E1 -22731.506,E2 -22731.506} C_VEL
LIN {X 0,Y 204.98,Z 460.623,A -85,B 0,C 180,E1 -22731.979,E2 -22731.979} C_VEL
LIN {X 0,Y 203.724,Z 481.872,A -85,B 0,C 180,E1 -22732.735,E2 -22732.735} C_VEL
LIN {X 0,Y 202.216,Z 494.501,A -85,B 0,C 180,E1 -22733.498,E2 -22733.498} C_VEL
LIN {X 0,Y 200.031,Z 506.765,A -85,B 0,C 180,E1 -22734.57,E2 -22734.57} C_VEL
LIN {X 0,Y 197.399,Z 518.01,A -85,B 0,C 180,E1 -22735.911,E2 -22735.911} C_VEL
LIN {X 0,Y 195.442,Z 523.226,A -85,B 0,C 180,E1 -22736.58,E2 -22736.58} C_VEL
LIN {X 0,Y 190.471,Z 531.239,A -85,B 0,C 180,E1 -22737.552,E2 -22737.552} C_VEL
LIN {X 0,Y 185.294,Z 538.664,A -85,B 0,C 180,E1 -22738.732,E2 -22738.732} C_VEL
LIN {X 0,Y 183.039,Z 543.012,A -85,B 0,C 180,E1 -22739.715,E2 -22739.715} C_VEL
LIN {X 0,Y 179.354,Z 552.662,A -85,B 0,C 180,E1 -22742.586,E2 -22742.586} C_VEL
LIN {X 0,Y 176.017,Z 561.095,A -85,B 0,C 180,E1 -22745.842,E2 -22745.842} C_VEL
LIN {X 0,Y 173.759,Z 566.897,A -85,B 0,C 180,E1 -22748.653,E2 -22748.653} C_VEL
LIN {X 0,Y 171.807,Z 572.627,A -85,B 0,C 180,E1 -22752.134,E2 -22752.134} C_VEL
LIN {X 0,Y 170.581,Z 577.18,A -85,B 0,C 180,E1 -22755.688,E2 -22755.688} C_VEL
LIN {X 0,Y 170.084,Z 580.676,A -85,B 0,C 180,E1 -22759.284,E2 -22759.284} C_VEL
LIN {X 0,Y 170.194,Z 583.186,A -85,B 0,C 180,E1 -22762.884,E2 -22762.884} C_VEL
LIN {X 0,Y 170.578,Z 584.327,A -85,B 0,C 180,E1 -22765.273,E2 -22765.273} C_VEL
LIN {X 0,Y 171.008,Z 585.048,A -85,B 0,C 180,E1 -22767.645,E2 -22767.645} C_VEL
LIN {X 0,Y 171.676,Z 585.369,A -85,B 0,C 180,E1 -22770,E2 -22770} C_VEL
LIN {X 0,Y 171.022,Z 585.037,A -85,B 0,C 180,E1 -22772.355,E2 -22772.355} C_VEL
LIN {X 0,Y 170.591,Z 584.308,A -85,B 0,C 180,E1 -22774.726,E2 -22774.726} C_VEL
LIN {X 0,Y 170.164,Z 582.897,A -85,B 0,C 180,E1 -22777.593,E2 -22777.593} C_VEL
LIN {X 0,Y 170.164,Z 579.568,A -85,B 0,C 180,E1 -22781.917,E2 -22781.917} C_VEL
LIN {X 0,Y 170.921,Z 575.712,A -85,B 0,C 180,E1 -22785.502,E2 -22785.502} C_VEL
LIN {X 0,Y 172.326,Z 570.747,A -85,B 0,C 180,E1 -22789.042,E2 -22789.042} C_VEL
LIN {X 0,Y 174.651,Z 564.574,A -85,B 0,C 180,E1 -22792.473,E2 -22792.473} C_VEL
LIN {X 0,Y 177.583,Z 556.931,A -85,B 0,C 180,E1 -22795.806,E2 -22795.806} C_VEL
LIN {X 0,Y 180.641,Z 549.204,A -85,B 0,C 180,E1 -22798.463,E2 -22798.463} C_VEL
LIN {X 0,Y 184.162,Z 539.887,A -85,B 0,C 180,E1 -22801.009,E2 -22801.009} C_VEL
LIN {X 0,Y 187.75,Z 529.566,A -85,B 0,C 180,E1 -22803.192,E2 -22803.192} C_VEL
LIN {X 0,Y 191.212,Z 518.152,A -85,B 0,C 180,E1 -22805.05,E2 -22805.05} C_VEL
LIN {X 0,Y 193.978,Z 506.281,A -85,B 0,C 180,E1 -22806.551,E2 -22806.551} C_VEL
LIN {X 0,Y 196.501,Z 493.135,A -85,B 0,C 180,E1 -22807.705,E2 -22807.705} C_VEL
LIN {X 0,Y 198.146,Z 479.514,A -85,B 0,C 180,E1 -22808.519,E2 -22808.519} C_VEL
LIN {X 0,Y 199.191,Z 460.31,A -85,B 0,C 180,E1 -22809.222,E2 -22809.222} C_VEL
LIN {X 0,Y 197.545,Z 430.233,A -85,B 0,C 180,E1 -22810.983,E2 -22810.983} C_VEL
LIN {X 0,Y 195.407,Z 404.564,A -85,B 0,C 180,E1 -22812.737,E2 -22812.737} C_VEL
LIN {X 0,Y 189.915,Z 391.484,A -85,B 0,C 180,E1 -22814.901,E2 -22814.901} C_VEL
LIN {X 0,Y 184.831,Z 380.851,A -85,B 0,C 180,E1 -22817.018,E2 -22817.018} C_VEL
LIN {X 0,Y 181.737,Z 374.993,A -85,B 0,C 180,E1 -22818.372,E2 -22818.372} C_VEL
LIN {X 0,Y 178.516,Z 369.154,A -85,B 0,C 180,E1 -22819.856,E2 -22819.856} C_VEL
LIN {X 0,Y 175.697,Z 363.73,A -85,B 0,C 180,E1 -22821.409,E2 -22821.409} C_VEL
LIN {X 0,Y 173.197,Z 355.481,A -85,B 0,C 180,E1 -22826.784,E2 -22826.784} C_VEL
LIN {X 0,Y 171.431,Z 350.191,A -85,B 0,C 180,E1 -22830.868,E2 -22830.868} C_VEL
LIN {X 0,Y 171.436,Z 350.121,A -85,B 0,C 180,E1 -22835.798,E2 -22835.798} C_VEL
LIN {X 0,Y 171.574,Z 350.072,A -85,B 0,C 180,E1 -22840.871,E2 -22840.871} C_VEL
LIN {X 0,Y 171.569,Z 350.093,A -85,B 0,C 180,E1 -22845.772,E2 -22845.772} C_VEL
LIN {X 0,Y 171.841,Z 350.08,A -85,B 0,C 180,E1 -22850.585,E2 -22850.585} C_VEL
LIN {X 0,Y 171.781,Z 350.067,A -85,B 0,C 180,E1 -22855.307,E2 -22855.307} C_VEL
LIN {X 0,Y 172.306,Z 349.995,A -85,B 0,C 180,E1 -22860,E2 -22860} C_VEL
LIN {X 0,Y 171.784,Z 350.086,A -85,B 0,C 180,E1 -22864.694,E2 -22864.694} C_VEL
LIN {X 0,Y 171.84,Z 350.059,A -85,B 0,C 180,E1 -22869.416,E2 -22869.416} C_VEL
LIN {X 0,Y 171.555,Z 350.088,A -85,B 0,C 180,E1 -22874.229,E2 -22874.229} C_VEL
LIN {X 0,Y 171.479,Z 350.108,A -85,B 0,C 180,E1 -22879.502,E2 -22879.502} C_VEL
LIN {X 0,Y 171.432,Z 350.102,A -85,B 0,C 180,E1 -22885.592,E2 -22885.592} C_VEL
LIN {X 0,Y 171.415,Z 350.056,A -85,B 0,C 180,E1 -22890.573,E2 -22890.573} C_VEL
LIN {X 0,Y 171.371,Z 350.104,A -85,B 0,C 180,E1 -22896.488,E2 -22896.488} C_VEL
LIN {X 0,Y 171.404,Z 350.442,A -85,B 0,C 180,E1 -22897.769,E2 -22897.769} C_VEL
LIN {X 0,Y 171.706,Z 351.529,A -85,B 0,C 180,E1 -22898.273,E2 -22898.273} C_VEL
LIN {X 0,Y 173.054,Z 353.883,A -85,B 0,C 180,E1 -22899.036,E2 -22899.036} C_VEL
LIN {X 0,Y 175.037,Z 355.666,A -85,B 0,C 180,E1 -22899.973,E2 -22899.973} C_VEL
LIN {X 0,Y 176.975,Z 358.852,A -85,B 0,C 180,E1 -22900.94,E2 -22900.94} C_VEL
LIN {X 0,Y 178.624,Z 360.798,A -85,B 0,C 180,E1 -22901.685,E2 -22901.685} C_VEL
LIN {X 0,Y 184.628,Z 369.413,A -85,B 0,C 180,E1 -22904.288,E2 -22904.288} C_VEL
LIN {X 0,Y 191.032,Z 379.302,A -85,B 0,C 180,E1 -22906.801,E2 -22906.801} C_VEL
LIN {X 0,Y 197.478,Z 390.717,A -85,B 0,C 180,E1 -22909.141,E2 -22909.141} C_VEL
LIN {X 0,Y 202.371,Z 400.652,A -85,B 0,C 180,E1 -22910.824,E2 -22910.824} C_VEL
LIN {X 0,Y 201.109,Z 435.987,A -85,B 0,C 180,E1 -22912.206,E2 -22912.206} C_VEL
LIN {X 0,Y 199.969,Z 449.331,A -85,B 0,C 180,E1 -22913.113,E2 -22913.113} C_VEL
LIN {X 0,Y 198.234,Z 461.996,A -85,B 0,C 180,E1 -22914.373,E2 -22914.373} C_VEL
LIN {X 0,Y 196.018,Z 473.342,A -85,B 0,C 180,E1 -22915.887,E2 -22915.887} C_VEL
LIN {X 0,Y 193.356,Z 483.514,A -85,B 0,C 180,E1 -22917.58,E2 -22917.58} C_VEL
LIN {X 0,Y 190.553,Z 492.791,A -85,B 0,C 180,E1 -22919.528,E2 -22919.528} C_VEL
LIN {X 0,Y 187.512,Z 502.235,A -85,B 0,C 180,E1 -22922.063,E2 -22922.063} C_VEL
LIN {X 0,Y 184.638,Z 509.971,A -85,B 0,C 180,E1 -22924.646,E2 -22924.646} C_VEL
LIN {X 0,Y 181.54,Z 517.626,A -85,B 0,C 180,E1 -22927.884,E2 -22927.884} C_VEL
LIN {X 0,Y 178.586,Z 524.425,A -85,B 0,C 180,E1 -22931.65,E2 -22931.65} C_VEL
LIN {X 0,Y 176.393,Z 529.032,A -85,B 0,C 180,E1 -22934.991,E2 -22934.991} C_VEL
LIN {X 0,Y 174.486,Z 532.577,A -85,B 0,C 180,E1 -22938.382,E2 -22938.382} C_VEL
LIN {X 0,Y 173.546,Z 534.399,A -85,B 0,C 180,E1 -22940.678,E2 -22940.678} C_VEL
LIN {X 0,Y 173.079,Z 535.731,A -85,B 0,C 180,E1 -22943.003,E2 -22943.003} C_VEL
LIN {X 0,Y 172.569,Z 536.702,A -85,B 0,C 180,E1 -22945.328,E2 -22945.328} C_VEL
LIN {X 0,Y 172.416,Z 537.277,A -85,B 0,C 180,E1 -22947.664,E2 -22947.664} C_VEL
LIN {X 0,Y 172.332,Z 537.499,A -85,B 0,C 180,E1 -22950,E2 -22950} C_VEL
LIN {X 0,Y 172.416,Z 537.309,A -85,B 0,C 180,E1 -22952.336,E2 -22952.336} C_VEL
LIN {X 0,Y 173.072,Z 535.804,A -85,B 0,C 180,E1 -22956.997,E2 -22956.997} C_VEL
LIN {X 0,Y 173.529,Z 534.506,A -85,B 0,C 180,E1 -22959.323,E2 -22959.323} C_VEL
LIN {X 0,Y 175.153,Z 531.664,A -85,B 0,C 180,E1 -22962.749,E2 -22962.749} C_VEL
LIN {X 0,Y 177.133,Z 527.829,A -85,B 0,C 180,E1 -22966.125,E2 -22966.125} C_VEL
LIN {X 0,Y 179.375,Z 522.741,A -85,B 0,C 180,E1 -22969.571,E2 -22969.571} C_VEL
LIN {X 0,Y 182.594,Z 515.49,A -85,B 0,C 180,E1 -22973.236,E2 -22973.236} C_VEL
LIN {X 0,Y 185.804,Z 507.454,A -85,B 0,C 180,E1 -22976.387,E2 -22976.387} C_VEL
LIN {X 0,Y 188.686,Z 499.222,A -85,B 0,C 180,E1 -22978.96,E2 -22978.96} C_VEL
LIN {X 0,Y 191.493,Z 490.178,A -85,B 0,C 180,E1 -22981.225,E2 -22981.225} C_VEL
LIN {X 0,Y 194.628,Z 479.627,A -85,B 0,C 180,E1 -22983.243,E2 -22983.243} C_VEL
LIN {X 0,Y 197.242,Z 468.085,A -85,B 0,C 180,E1 -22985.008,E2 -22985.008} C_VEL
LIN {X 0,Y 199.316,Z 456.776,A -85,B 0,C 180,E1 -22986.309,E2 -22986.309} C_VEL
LIN {X 0,Y 200.694,Z 443.891,A -85,B 0,C 180,E1 -22987.44,E2 -22987.44} C_VEL
LIN {X 0,Y 201.419,Z 431.092,A -85,B 0,C 180,E1 -22988.181,E2 -22988.181} C_VEL
LIN {X 0,Y 202.519,Z 400.837,A -85,B 0,C 180,E1 -22989.307,E2 -22989.307} C_VEL
LIN {X 0,Y 196.043,Z 387.944,A -85,B 0,C 180,E1 -22991.554,E2 -22991.554} C_VEL
LIN {X 0,Y 189.881,Z 377.479,A -85,B 0,C 180,E1 -22993.826,E2 -22993.826} C_VEL
LIN {X 0,Y 183.727,Z 368.012,A -85,B 0,C 180,E1 -22996.294,E2 -22996.294} C_VEL
LIN {X 0,Y 180.527,Z 363.603,A -85,B 0,C 180,E1 -22997.664,E2 -22997.664} C_VEL
LIN {X 0,Y 177.807,Z 359.692,A -85,B 0,C 180,E1 -22998.908,E2 -22998.908} C_VEL
LIN {X 0,Y 175.585,Z 356.8,A -85,B 0,C 180,E1 -22999.96,E2 -22999.96} C_VEL
LIN {X 0,Y 174.752,Z 355.334,A -85,B 0,C 180,E1 -23000.391,E2 -23000.391} C_VEL
LIN {X 0,Y 172.412,Z 353.039,A -85,B 0,C 180,E1 -23001.528,E2 -23001.528} C_VEL
LIN {X 0,Y 171.492,Z 350.75,A -85,B 0,C 180,E1 -23002.254,E2 -23002.254} C_VEL
LIN {X 0,Y 171.354,Z 350.148,A -85,B 0,C 180,E1 -23003.141,E2 -23003.141} C_VEL
LIN {X 0,Y 171.391,Z 350.079,A -85,B 0,C 180,E1 -23007.786,E2 -23007.786} C_VEL
LIN {X 0,Y 171.405,Z 350.054,A -85,B 0,C 180,E1 -23010.526,E2 -23010.526} C_VEL
LIN {X 0,Y 171.424,Z 350.132,A -85,B 0,C 180,E1 -23015.796,E2 -23015.796} C_VEL
LIN {X 0,Y 171.504,Z 350.109,A -85,B 0,C 180,E1 -23020.863,E2 -23020.863} C_VEL
LIN {X 0,Y 171.549,Z 350.09,A -85,B 0,C 180,E1 -23025.77,E2 -23025.77} C_VEL
LIN {X 0,Y 171.84,Z 350.061,A -85,B 0,C 180,E1 -23030.584,E2 -23030.584} C_VEL
LIN {X 0,Y 171.783,Z 350.088,A -85,B 0,C 180,E1 -23035.306,E2 -23035.306} C_VEL
LIN {X 0,Y 172.305,Z 349.995,A -85,B 0,C 180,E1 -23040,E2 -23040} C_VEL
LIN {X 0,Y 171.779,Z 350.065,A -85,B 0,C 180,E1 -23044.693,E2 -23044.693} C_VEL
LIN {X 0,Y 171.84,Z 350.079,A -85,B 0,C 180,E1 -23049.415,E2 -23049.415} C_VEL
LIN {X 0,Y 171.563,Z 350.095,A -85,B 0,C 180,E1 -23054.228,E2 -23054.228} C_VEL
LIN {X 0,Y 171.524,Z 350.073,A -85,B 0,C 180,E1 -23059.545,E2 -23059.545} C_VEL
LIN {X 0,Y 171.44,Z 350.119,A -85,B 0,C 180,E1 -23065.597,E2 -23065.597} C_VEL
LIN {X 0,Y 171.428,Z 350.327,A -85,B 0,C 180,E1 -23069.133,E2 -23069.133} C_VEL
LIN {X 0,Y 173.214,Z 355.67,A -85,B 0,C 180,E1 -23073.213,E2 -23073.213} C_VEL
LIN {X 0,Y 175.597,Z 363.462,A -85,B 0,C 180,E1 -23078.343,E2 -23078.343} C_VEL
LIN {X 0,Y 176.712,Z 366.049,A -85,B 0,C 180,E1 -23079.151,E2 -23079.151} C_VEL
LIN {X 0,Y 180.162,Z 371.93,A -85,B 0,C 180,E1 -23080.783,E2 -23080.783} C_VEL
LIN {X 0,Y 184.23,Z 379.687,A -85,B 0,C 180,E1 -23082.613,E2 -23082.613} C_VEL
LIN {X 0,Y 189.339,Z 390.073,A -85,B 0,C 180,E1 -23084.756,E2 -23084.756} C_VEL
LIN {X 0,Y 194.549,Z 402.262,A -85,B 0,C 180,E1 -23086.832,E2 -23086.832} C_VEL
LIN {X 0,Y 195.489,Z 404.856,A -85,B 0,C 180,E1 -23087.207,E2 -23087.207} C_VEL
LIN {X 0,Y 197.192,Z 424.392,A -85,B 0,C 180,E1 -23088.571,E2 -23088.571} C_VEL
LIN {X 0,Y 199.048,Z 453.334,A -85,B 0,C 180,E1 -23090.348,E2 -23090.348} C_VEL
LIN {X 0,Y 199.248,Z 462.424,A -85,B 0,C 180,E1 -23090.804,E2 -23090.804} C_VEL
LIN {X 0,Y 198.077,Z 481.063,A -85,B 0,C 180,E1 -23091.493,E2 -23091.493} C_VEL
LIN {X 0,Y 196.407,Z 494.384,A -85,B 0,C 180,E1 -23092.325,E2 -23092.325} C_VEL
LIN {X 0,Y 194.054,Z 506.796,A -85,B 0,C 180,E1 -23093.466,E2 -23093.466} C_VEL
LIN {X 0,Y 191.138,Z 518.528,A -85,B 0,C 180,E1 -23094.935,E2 -23094.935} C_VEL
LIN {X 0,Y 187.751,Z 529.884,A -85,B 0,C 180,E1 -23096.808,E2 -23096.808} C_VEL
LIN {X 0,Y 184.165,Z 540.133,A -85,B 0,C 180,E1 -23098.991,E2 -23098.991} C_VEL
LIN {X 0,Y 183.039,Z 543.012,A -85,B 0,C 180,E1 -23099.715,E2 -23099.715} C_VEL
LIN {X 0,Y 180.78,Z 547.273,A -85,B 0,C 180,E1 -23100.798,E2 -23100.798} C_VEL
LIN {X 0,Y 175.513,Z 553.681,A -85,B 0,C 180,E1 -23102.558,E2 -23102.558} C_VEL
LIN {X 0,Y 170.404,Z 559.481,A -85,B 0,C 180,E1 -23104.609,E2 -23104.609} C_VEL
LIN {X 0,Y 168.44,Z 562.782,A -85,B 0,C 180,E1 -23106.122,E2 -23106.122} C_VEL
LIN {X 0,Y 166.226,Z 567.963,A -85,B 0,C 180,E1 -23108.938,E2 -23108.938} C_VEL
LIN {X 0,Y 164.467,Z 573.294,A -85,B 0,C 180,E1 -23112.595,E2 -23112.595} C_VEL
LIN {X 0,Y 163.372,Z 577.484,A -85,B 0,C 180,E1 -23116.314,E2 -23116.314} C_VEL
LIN {X 0,Y 162.986,Z 580.645,A -85,B 0,C 180,E1 -23120.068,E2 -23120.068} C_VEL
LIN {X 0,Y 163.141,Z 582.198,A -85,B 0,C 180,E1 -23122.575,E2 -23122.575} C_VEL
LIN {X 0,Y 163.489,Z 583.338,A -85,B 0,C 180,E1 -23125.068,E2 -23125.068} C_VEL
LIN {X 0,Y 163.925,Z 584.062,A -85,B 0,C 180,E1 -23127.543,E2 -23127.543} C_VEL
LIN {X 0,Y 164.593,Z 584.384,A -85,B 0,C 180,E1 -23130,E2 -23130} C_VEL
LIN {X 0,Y 163.938,Z 584.05,A -85,B 0,C 180,E1 -23132.457,E2 -23132.457} C_VEL
LIN {X 0,Y 163.5,Z 583.317,A -85,B 0,C 180,E1 -23134.932,E2 -23134.932} C_VEL
LIN {X 0,Y 163.094,Z 582.052,A -85,B 0,C 180,E1 -23137.644,E2 -23137.644} C_VEL
LIN {X 0,Y 163.049,Z 579.629,A -85,B 0,C 180,E1 -23141.184,E2 -23141.184} C_VEL
LIN {X 0,Y 163.632,Z 576.107,A -85,B 0,C 180,E1 -23144.933,E2 -23144.933} C_VEL
LIN {X 0,Y 164.976,Z 571.529,A -85,B 0,C 180,E1 -23148.632,E2 -23148.632} C_VEL
LIN {X 0,Y 167.354,Z 565.319,A -85,B 0,C 180,E1 -23152.499,E2 -23152.499} C_VEL
LIN {X 0,Y 170.597,Z 557.32,A -85,B 0,C 180,E1 -23156.286,E2 -23156.286} C_VEL
LIN {X 0,Y 174.409,Z 548.21,A -85,B 0,C 180,E1 -23159.579,E2 -23159.579} C_VEL
LIN {X 0,Y 178.113,Z 538.896,A -85,B 0,C 180,E1 -23162.186,E2 -23162.186} C_VEL
LIN {X 0,Y 181.824,Z 528.57,A -85,B 0,C 180,E1 -23164.422,E2 -23164.422} C_VEL
LIN {X 0,Y 185.417,Z 517.154,A -85,B 0,C 180,E1 -23166.316,E2 -23166.316} C_VEL
LIN {X 0,Y 188.334,Z 505.289,A -85,B 0,C 180,E1 -23167.834,E2 -23167.834} C_VEL
LIN {X 0,Y 190.896,Z 492.349,A -85,B 0,C 180,E1 -23168.993,E2 -23168.993} C_VEL
LIN {X 0,Y 192.627,Z 478.474,A -85,B 0,C 180,E1 -23169.841,E2 -23169.841} C_VEL
LIN {X 0,Y 193.627,Z 460.569,A -85,B 0,C 180,E1 -23170.519,E2 -23170.519} C_VEL
LIN {X 0,Y 192.127,Z 431.251,A -85,B 0,C 180,E1 -23172.302,E2 -23172.302} C_VEL
LIN {X 0,Y 190.253,Z 407.29,A -85,B 0,C 180,E1 -23173.999,E2 -23173.999} C_VEL
LIN {X 0,Y 185.26,Z 395.128,A -85,B 0,C 180,E1 -23176.107,E2 -23176.107} C_VEL
LIN {X 0,Y 180.177,Z 384.406,A -85,B 0,C 180,E1 -23178.368,E2 -23178.368} C_VEL
LIN {X 0,Y 177.281,Z 378.853,A -85,B 0,C 180,E1 -23179.728,E2 -23179.728} C_VEL
LIN {X 0,Y 174.755,Z 374.105,A -85,B 0,C 180,E1 -23180.977,E2 -23180.977} C_VEL
LIN {X 0,Y 171.412,Z 368.166,A -85,B 0,C 180,E1 -23182.718,E2 -23182.718} C_VEL
LIN {X 0,Y 167.956,Z 362.118,A -85,B 0,C 180,E1 -23184.784,E2 -23184.784} C_VEL
LIN {X 0,Y 166.229,Z 356.663,A -85,B 0,C 180,E1 -23188.687,E2 -23188.687} C_VEL
LIN {X 0,Y 164.362,Z 351.084,A -85,B 0,C 180,E1 -23193.45,E2 -23193.45} C_VEL
LIN {X 0,Y 164.47,Z 350.949,A -85,B 0,C 180,E1 -23200.01,E2 -23200.01} C_VEL
LIN {X 0,Y 164.5,Z 350.979,A -85,B 0,C 180,E1 -23205.147,E2 -23205.147} C_VEL
LIN {X 0,Y 164.763,Z 350.962,A -85,B 0,C 180,E1 -23210.176,E2 -23210.176} C_VEL
LIN {X 0,Y 164.819,Z 350.931,A -85,B 0,C 180,E1 -23212.651,E2 -23212.651} C_VEL
LIN {X 0,Y 165.27,Z 350.871,A -85,B 0,C 180,E1 -23220,E2 -23220} C_VEL
LIN {X 0,Y 164.816,Z 350.926,A -85,B 0,C 180,E1 -23227.35,E2 -23227.35} C_VEL
LIN {X 0,Y 164.699,Z 350.968,A -85,B 0,C 180,E1 -23231.058,E2 -23231.058} C_VEL
LIN {X 0,Y 164.439,Z 351,A -85,B 0,C 180,E1 -23237.408,E2 -23237.408} C_VEL
LIN {X 0,Y 164.345,Z 350.998,A -85,B 0,C 180,E1 -23242.636,E2 -23242.636} C_VEL
LIN {X 0,Y 164.36,Z 350.968,A -85,B 0,C 180,E1 -23246.112,E2 -23246.112} C_VEL
LIN {X 0,Y 164.35,Z 350.94,A -85,B 0,C 180,E1 -23251.215,E2 -23251.215} C_VEL
LIN {X 0,Y 164.377,Z 351.307,A -85,B 0,C 180,E1 -23254.388,E2 -23254.388} C_VEL
LIN {X 0,Y 164.676,Z 352.372,A -85,B 0,C 180,E1 -23254.992,E2 -23254.992} C_VEL
LIN {X 0,Y 166.082,Z 354.829,A -85,B 0,C 180,E1 -23255.917,E2 -23255.917} C_VEL
LIN {X 0,Y 168.244,Z 356.716,A -85,B 0,C 180,E1 -23257.092,E2 -23257.092} C_VEL
LIN {X 0,Y 170.288,Z 359.98,A -85,B 0,C 180,E1 -23258.249,E2 -23258.249} C_VEL
LIN {X 0,Y 172.032,Z 361.903,A -85,B 0,C 180,E1 -23259.133,E2 -23259.133} C_VEL
LIN {X 0,Y 178.76,Z 371.457,A -85,B 0,C 180,E1 -23262.374,E2 -23262.374} C_VEL
LIN {X 0,Y 185.324,Z 381.462,A -85,B 0,C 180,E1 -23265.176,E2 -23265.176} C_VEL
LIN {X 0,Y 191.958,Z 393.115,A -85,B 0,C 180,E1 -23267.768,E2 -23267.768} C_VEL
LIN {X 0,Y 196.975,Z 403.399,A -85,B 0,C 180,E1 -23269.616,E2 -23269.616} C_VEL
LIN {X 0,Y 195.557,Z 437.446,A -85,B 0,C 180,E1 -23270.967,E2 -23270.967} C_VEL
LIN {X 0,Y 194.315,Z 451.035,A -85,B 0,C 180,E1 -23271.93,E2 -23271.93} C_VEL
LIN {X 0,Y 192.565,Z 462.981,A -85,B 0,C 180,E1 -23273.154,E2 -23273.154} C_VEL
LIN {X 0,Y 190.019,Z 475.3,A -85,B 0,C 180,E1 -23274.856,E2 -23274.856} C_VEL
LIN {X 0,Y 187.095,Z 485.767,A -85,B 0,C 180,E1 -23276.677,E2 -23276.677} C_VEL
LIN {X 0,Y 184.221,Z 494.817,A -85,B 0,C 180,E1 -23278.682,E2 -23278.682} C_VEL
LIN {X 0,Y 181.332,Z 503.216,A -85,B 0,C 180,E1 -23281.023,E2 -23281.023} C_VEL
LIN {X 0,Y 178.312,Z 510.951,A -85,B 0,C 180,E1 -23283.679,E2 -23283.679} C_VEL
LIN {X 0,Y 175.049,Z 518.605,A -85,B 0,C 180,E1 -23287.018,E2 -23287.018} C_VEL
LIN {X 0,Y 171.929,Z 525.405,A -85,B 0,C 180,E1 -23290.912,E2 -23290.912} C_VEL
LIN {X 0,Y 169.615,Z 530.011,A -85,B 0,C 180,E1 -23294.376,E2 -23294.376} C_VEL
LIN {X 0,Y 167.605,Z 533.556,A -85,B 0,C 180,E1 -23297.898,E2 -23297.898} C_VEL
LIN {X 0,Y 166.611,Z 535.378,A -85,B 0,C 180,E1 -23300.286,E2 -23300.286} C_VEL
LIN {X 0,Y 166.104,Z 536.709,A -85,B 0,C 180,E1 -23302.708,E2 -23302.708} C_VEL
LIN {X 0,Y 165.394,Z 538.256,A -85,B 0,C 180,E1 -23307.565,E2 -23307.565} C_VEL
LIN {X 0,Y 165.304,Z 538.477,A -85,B 0,C 180,E1 -23310,E2 -23310} C_VEL
LIN {X 0,Y 165.394,Z 538.287,A -85,B 0,C 180,E1 -23312.435,E2 -23312.435} C_VEL
LIN {X 0,Y 166.096,Z 536.781,A -85,B 0,C 180,E1 -23317.293,E2 -23317.293} C_VEL
LIN {X 0,Y 166.594,Z 535.484,A -85,B 0,C 180,E1 -23319.715,E2 -23319.715} C_VEL
LIN {X 0,Y 168.305,Z 532.641,A -85,B 0,C 180,E1 -23323.277,E2 -23323.277} C_VEL
LIN {X 0,Y 170.392,Z 528.806,A -85,B 0,C 180,E1 -23326.781,E2 -23326.781} C_VEL
LIN {X 0,Y 172.769,Z 523.717,A -85,B 0,C 180,E1 -23330.352,E2 -23330.352} C_VEL
LIN {X 0,Y 176.157,Z 516.466,A -85,B 0,C 180,E1 -23334.138,E2 -23334.138} C_VEL
LIN {X 0,Y 179.535,Z 508.43,A -85,B 0,C 180,E1 -23337.384,E2 -23337.384} C_VEL
LIN {X 0,Y 182.566,Z 500.197,A -85,B 0,C 180,E1 -23340.029,E2 -23340.029} C_VEL
LIN {X 0,Y 185.509,Z 491.154,A -85,B 0,C 180,E1 -23342.352,E2 -23342.352} C_VEL
LIN {X 0,Y 188.792,Z 480.6,A -85,B 0,C 180,E1 -23344.412,E2 -23344.412} C_VEL
LIN {X 0,Y 191.528,Z 469.057,A -85,B 0,C 180,E1 -23346.215,E2 -23346.215} C_VEL
LIN {X 0,Y 193.693,Z 457.747,A -85,B 0,C 180,E1 -23347.542,E2 -23347.542} C_VEL
LIN {X 0,Y 195.152,Z 444.803,A -85,B 0,C 180,E1 -23348.701,E2 -23348.701} C_VEL
LIN {X 0,Y 195.94,Z 432.437,A -85,B 0,C 180,E1 -23349.431,E2 -23349.431} C_VEL
LIN {X 0,Y 197.011,Z 403.139,A -85,B 0,C 180,E1 -23350.567,E2 -23350.567} C_VEL
LIN {X 0,Y 190.414,Z 390.069,A -85,B 0,C 180,E1 -23353.017,E2 -23353.017} C_VEL
LIN {X 0,Y 182.876,Z 377.49,A -85,B 0,C 180,E1 -23356.046,E2 -23356.046} C_VEL
LIN {X 0,Y 177.278,Z 369.322,A -85,B 0,C 180,E1 -23358.52,E2 -23358.52} C_VEL
LIN {X 0,Y 174.35,Z 365.188,A -85,B 0,C 180,E1 -23359.922,E2 -23359.922} C_VEL
LIN {X 0,Y 171.426,Z 361.102,A -85,B 0,C 180,E1 -23361.414,E2 -23361.414} C_VEL
LIN {X 0,Y 168.963,Z 358.136,A -85,B 0,C 180,E1 -23362.719,E2 -23362.719} C_VEL
LIN {X 0,Y 168.094,Z 356.447,A -85,B 0,C 180,E1 -23363.244,E2 -23363.244} C_VEL
LIN {X 0,Y 165.697,Z 354.387,A -85,B 0,C 180,E1 -23364.564,E2 -23364.564} C_VEL
LIN {X 0,Y 164.438,Z 351.608,A -85,B 0,C 180,E1 -23365.627,E2 -23365.627} C_VEL
LIN {X 0,Y 164.309,Z 351.038,A -85,B 0,C 180,E1 -23366.57,E2 -23366.57} C_VEL
LIN {X 0,Y 164.364,Z 350.935,A -85,B 0,C 180,E1 -23369.129,E2 -23369.129} C_VEL
LIN {X 0,Y 164.383,Z 350.983,A -85,B 0,C 180,E1 -23374.688,E2 -23374.688} C_VEL
LIN {X 0,Y 164.414,Z 350.985,A -85,B 0,C 180,E1 -23380.117,E2 -23380.117} C_VEL
LIN {X 0,Y 164.478,Z 350.97,A -85,B 0,C 180,E1 -23385.145,E2 -23385.145} C_VEL
LIN {X 0,Y 164.761,Z 350.946,A -85,B 0,C 180,E1 -23390.176,E2 -23390.176} C_VEL
LIN {X 0,Y 164.816,Z 350.928,A -85,B 0,C 180,E1 -23392.65,E2 -23392.65} C_VEL
LIN {X 0,Y 165.27,Z 350.871,A -85,B 0,C 180,E1 -23400,E2 -23400} C_VEL
LIN {X 0,Y 164.816,Z 350.931,A -85,B 0,C 180,E1 -23407.35,E2 -23407.35} C_VEL
LIN {X 0,Y 164.699,Z 350.952,A -85,B 0,C 180,E1 -23411.058,E2 -23411.058} C_VEL
LIN {X 0,Y 164.468,Z 350.98,A -85,B 0,C 180,E1 -23417.405,E2 -23417.405} C_VEL
LIN {X 0,Y 164.449,Z 350.951,A -85,B 0,C 180,E1 -23419.992,E2 -23419.992} C_VEL
LIN {X 0,Y 164.379,Z 351.127,A -85,B 0,C 180,E1 -23426.479,E2 -23426.479} C_VEL
LIN {X 0,Y 166.306,Z 356.935,A -85,B 0,C 180,E1 -23431.386,E2 -23431.386} C_VEL
LIN {X 0,Y 168,Z 362.204,A -85,B 0,C 180,E1 -23435.114,E2 -23435.114} C_VEL
LIN {X 0,Y 171.711,Z 368.554,A -85,B 0,C 180,E1 -23437.293,E2 -23437.293} C_VEL
LIN {X 0,Y 176.386,Z 376.985,A -85,B 0,C 180,E1 -23439.699,E2 -23439.699} C_VEL
LIN {X 0,Y 179.872,Z 383.731,A -85,B 0,C 180,E1 -23441.369,E2 -23441.369} C_VEL
LIN {X 0,Y 184.422,Z 393.124,A -85,B 0,C 180,E1 -23443.413,E2 -23443.413} C_VEL
LIN {X 0,Y 189.465,Z 405.072,A -85,B 0,C 180,E1 -23445.566,E2 -23445.566} C_VEL
LIN {X 0,Y 190.412,Z 407.803,A -85,B 0,C 180,E1 -23445.974,E2 -23445.974} C_VEL
LIN {X 0,Y 192.308,Z 431.953,A -85,B 0,C 180,E1 -23447.687,E2 -23447.687} C_VEL
LIN {X 0,Y 193.75,Z 461.004,A -85,B 0,C 180,E1 -23449.444,E2 -23449.444} C_VEL
LIN {X 0,Y 192.631,Z 479.697,A -85,B 0,C 180,E1 -23450.163,E2 -23450.163} C_VEL
LIN {X 0,Y 190.899,Z 492.953,A -85,B 0,C 180,E1 -23450.987,E2 -23450.987} C_VEL
LIN {X 0,Y 188.357,Z 505.807,A -85,B 0,C 180,E1 -23452.171,E2 -23452.171} C_VEL
LIN {X 0,Y 185.341,Z 517.54,A -85,B 0,C 180,E1 -23453.667,E2 -23453.667} C_VEL
LIN {X 0,Y 181.826,Z 528.895,A -85,B 0,C 180,E1 -23455.578,E2 -23455.578} C_VEL
LIN {X 0,Y 178.115,Z 539.147,A -85,B 0,C 180,E1 -23457.814,E2 -23457.814} C_VEL
LIN {X 0,Y 174.393,Z 548.409,A -85,B 0,C 180,E1 -23460.418,E2 -23460.418} C_VEL
LIN {X 0,Y 170.606,Z 557.488,A -85,B 0,C 180,E1 -23463.715,E2 -23463.715} C_VEL
LIN {X 0,Y 168.44,Z 562.782,A -85,B 0,C 180,E1 -23466.122,E2 -23466.122} C_VEL
LIN {X 0,Y 166.937,Z 564.914,A -85,B 0,C 180,E1 -23467.17,E2 -23467.17} C_VEL
LIN {X 0,Y 162.859,Z 567.865,A -85,B 0,C 180,E1 -23468.748,E2 -23468.748} C_VEL
LIN {X 0,Y 158.927,Z 570.519,A -85,B 0,C 180,E1 -23470.459,E2 -23470.459} C_VEL
LIN {X 0,Y 157.68,Z 572.13,A -85,B 0,C 180,E1 -23471.687,E2 -23471.687} C_VEL
LIN {X 0,Y 156.4,Z 576.485,A -85,B 0,C 180,E1 -23475.691,E2 -23475.691} C_VEL
LIN {X 0,Y 155.941,Z 579.65,A -85,B 0,C 180,E1 -23479.615,E2 -23479.615} C_VEL
LIN {X 0,Y 156.387,Z 582.346,A -85,B 0,C 180,E1 -23484.843,E2 -23484.843} C_VEL
LIN {X 0,Y 156.843,Z 583.075,A -85,B 0,C 180,E1 -23487.432,E2 -23487.432} C_VEL
LIN {X 0,Y 157.51,Z 583.398,A -85,B 0,C 180,E1 -23490,E2 -23490} C_VEL
LIN {X 0,Y 156.855,Z 583.063,A -85,B 0,C 180,E1 -23492.568,E2 -23492.568} C_VEL
LIN {X 0,Y 156.395,Z 582.325,A -85,B 0,C 180,E1 -23495.156,E2 -23495.156} C_VEL
LIN {X 0,Y 156.03,Z 581.169,A -85,B 0,C 180,E1 -23497.766,E2 -23497.766} C_VEL
LIN {X 0,Y 156.021,Z 578.631,A -85,B 0,C 180,E1 -23501.695,E2 -23501.695} C_VEL
LIN {X 0,Y 156.715,Z 575.108,A -85,B 0,C 180,E1 -23505.609,E2 -23505.609} C_VEL
LIN {X 0,Y 158.174,Z 570.526,A -85,B 0,C 180,E1 -23509.465,E2 -23509.465} C_VEL
LIN {X 0,Y 160.571,Z 564.792,A -85,B 0,C 180,E1 -23513.198,E2 -23513.198} C_VEL
LIN {X 0,Y 163.639,Z 557.688,A -85,B 0,C 180,E1 -23516.804,E2 -23516.804} C_VEL
LIN {X 0,Y 166.816,Z 550.492,A -85,B 0,C 180,E1 -23519.671,E2 -23519.671} C_VEL
LIN {X 0,Y 170.456,Z 541.849,A -85,B 0,C 180,E1 -23522.411,E2 -23522.411} C_VEL
LIN {X 0,Y 174.256,Z 532.428,A -85,B 0,C 180,E1 -23524.727,E2 -23524.727} C_VEL
LIN {X 0,Y 178.358,Z 520.771,A -85,B 0,C 180,E1 -23526.934,E2 -23526.934} C_VEL
LIN {X 0,Y 181.578,Z 509.263,A -85,B 0,C 180,E1 -23528.617,E2 -23528.617} C_VEL
LIN {X 0,Y 184.319,Z 497.431,A -85,B 0,C 180,E1 -23529.87,E2 -23529.87} C_VEL
LIN {X 0,Y 186.486,Z 483.901,A -85,B 0,C 180,E1 -23530.892,E2 -23530.892} C_VEL
LIN {X 0,Y 187.726,Z 470.731,A -85,B 0,C 180,E1 -23531.518,E2 -23531.518} C_VEL
LIN {X 0,Y 188.152,Z 460.336,A -85,B 0,C 180,E1 -23531.919,E2 -23531.919} C_VEL
LIN {X 0,Y 186.823,Z 432.46,A -85,B 0,C 180,E1 -23533.685,E2 -23533.685} C_VEL
LIN {X 0,Y 185.228,Z 410.009,A -85,B 0,C 180,E1 -23535.322,E2 -23535.322} C_VEL
LIN {X 0,Y 179.557,Z 396.175,A -85,B 0,C 180,E1 -23537.904,E2 -23537.904} C_VEL
LIN {X 0,Y 174.397,Z 385.352,A -85,B 0,C 180,E1 -23540.415,E2 -23540.415} C_VEL
LIN {X 0,Y 170.667,Z 378.348,A -85,B 0,C 180,E1 -23542.359,E2 -23542.359} C_VEL
LIN {X 0,Y 167.862,Z 373.228,A -85,B 0,C 180,E1 -23543.927,E2 -23543.927} C_VEL
LIN {X 0,Y 163.875,Z 366.523,A -85,B 0,C 180,E1 -23546.316,E2 -23546.316} C_VEL
LIN {X 0,Y 160.139,Z 360.203,A -85,B 0,C 180,E1 -23548.958,E2 -23548.958} C_VEL
LIN {X 0,Y 158.667,Z 356.101,A -85,B 0,C 180,E1 -23552.358,E2 -23552.358} C_VEL
LIN {X 0,Y 157.321,Z 351.942,A -85,B 0,C 180,E1 -23556.468,E2 -23556.468} C_VEL
LIN {X 0,Y 157.4,Z 351.846,A -85,B 0,C 180,E1 -23561.787,E2 -23561.787} C_VEL
LIN {X 0,Y 157.512,Z 351.838,A -85,B 0,C 180,E1 -23567.109,E2 -23567.109} C_VEL
LIN {X 0,Y 157.685,Z 351.838,A -85,B 0,C 180,E1 -23569.731,E2 -23569.731} C_VEL
LIN {X 0,Y 157.757,Z 351.813,A -85,B 0,C 180,E1 -23572.32,E2 -23572.32} C_VEL
LIN {X 0,Y 158.232,Z 351.747,A -85,B 0,C 180,E1 -23580,E2 -23580} C_VEL
LIN {X 0,Y 157.755,Z 351.805,A -85,B 0,C 180,E1 -23587.681,E2 -23587.681} C_VEL
LIN {X 0,Y 157.629,Z 351.849,A -85,B 0,C 180,E1 -23591.227,E2 -23591.227} C_VEL
LIN {X 0,Y 157.416,Z 351.851,A -85,B 0,C 180,E1 -23595.538,E2 -23595.538} C_VEL
LIN {X 0,Y 157.306,Z 351.866,A -85,B 0,C 180,E1 -23600.942,E2 -23600.942} C_VEL
LIN {X 0,Y 157.29,Z 351.835,A -85,B 0,C 180,E1 -23606.668,E2 -23606.668} C_VEL
LIN {X 0,Y 157.323,Z 352.138,A -85,B 0,C 180,E1 -23610.329,E2 -23610.329} C_VEL
LIN {X 0,Y 157.665,Z 353.268,A -85,B 0,C 180,E1 -23611.088,E2 -23611.088} C_VEL
LIN {X 0,Y 159.069,Z 355.787,A -85,B 0,C 180,E1 -23612.196,E2 -23612.196} C_VEL
LIN {X 0,Y 161.545,Z 357.841,A -85,B 0,C 180,E1 -23613.783,E2 -23613.783} C_VEL
LIN {X 0,Y 163.411,Z 360.906,A -85,B 0,C 180,E1 -23615.022,E2 -23615.022} C_VEL
LIN {X 0,Y 165.437,Z 362.987,A -85,B 0,C 180,E1 -23616.202,E2 -23616.202} C_VEL
LIN {X 0,Y 168.024,Z 366.572,A -85,B 0,C 180,E1 -23617.686,E2 -23617.686} C_VEL
LIN {X 0,Y 172.702,Z 373.152,A -85,B 0,C 180,E1 -23620.147,E2 -23620.147} C_VEL
LIN {X 0,Y 177.821,Z 380.775,A -85,B 0,C 180,E1 -23622.588,E2 -23622.588} C_VEL
LIN {X 0,Y 183.705,Z 390.435,A -85,B 0,C 180,E1 -23625.15,E2 -23625.15} C_VEL
LIN {X 0,Y 189.097,Z 400.569,A -85,B 0,C 180,E1 -23627.332,E2 -23627.332} C_VEL
LIN {X 0,Y 191.554,Z 405.562,A -85,B 0,C 180,E1 -23628.28,E2 -23628.28} C_VEL
LIN {X 0,Y 190.157,Z 438.374,A -85,B 0,C 180,E1 -23629.631,E2 -23629.631} C_VEL
LIN {X 0,Y 188.877,Z 451.552,A -85,B 0,C 180,E1 -23630.572,E2 -23630.572} C_VEL
LIN {X 0,Y 186.988,Z 463.965,A -85,B 0,C 180,E1 -23631.863,E2 -23631.863} C_VEL
LIN {X 0,Y 184.314,Z 476.286,A -85,B 0,C 180,E1 -23633.598,E2 -23633.598} C_VEL
LIN {X 0,Y 181.264,Z 486.75,A -85,B 0,C 180,E1 -23635.456,E2 -23635.456} C_VEL
LIN {X 0,Y 178.252,Z 495.799,A -85,B 0,C 180,E1 -23637.508,E2 -23637.508} C_VEL
LIN {X 0,Y 175.216,Z 504.197,A -85,B 0,C 180,E1 -23639.909,E2 -23639.909} C_VEL
LIN {X 0,Y 172.041,Z 511.932,A -85,B 0,C 180,E1 -23642.641,E2 -23642.641} C_VEL
LIN {X 0,Y 168.601,Z 519.585,A -85,B 0,C 180,E1 -23646.086,E2 -23646.086} C_VEL
LIN {X 0,Y 165.304,Z 526.384,A -85,B 0,C 180,E1 -23650.116,E2 -23650.116} C_VEL
LIN {X 0,Y 162.857,Z 530.99,A -85,B 0,C 180,E1 -23653.71,E2 -23653.71} C_VEL
LIN {X 0,Y 160.737,Z 534.535,A -85,B 0,C 180,E1 -23657.372,E2 -23657.372} C_VEL
LIN {X 0,Y 159.685,Z 536.357,A -85,B 0,C 180,E1 -23659.861,E2 -23659.861} C_VEL
LIN {X 0,Y 159.133,Z 537.688,A -85,B 0,C 180,E1 -23662.387,E2 -23662.387} C_VEL
LIN {X 0,Y 158.373,Z 539.234,A -85,B 0,C 180,E1 -23667.457,E2 -23667.457} C_VEL
LIN {X 0,Y 158.276,Z 539.455,A -85,B 0,C 180,E1 -23670,E2 -23670} C_VEL
LIN {X 0,Y 158.372,Z 539.265,A -85,B 0,C 180,E1 -23672.543,E2 -23672.543} C_VEL
LIN {X 0,Y 159.126,Z 537.759,A -85,B 0,C 180,E1 -23677.614,E2 -23677.614} C_VEL
LIN {X 0,Y 159.667,Z 536.462,A -85,B 0,C 180,E1 -23680.141,E2 -23680.141} C_VEL
LIN {X 0,Y 161.473,Z 533.618,A -85,B 0,C 180,E1 -23683.85,E2 -23683.85} C_VEL
LIN {X 0,Y 163.676,Z 529.783,A -85,B 0,C 180,E1 -23687.491,E2 -23687.491} C_VEL
LIN {X 0,Y 166.198,Z 524.693,A -85,B 0,C 180,E1 -23691.194,E2 -23691.194} C_VEL
LIN {X 0,Y 169.768,Z 517.442,A -85,B 0,C 180,E1 -23695.108,E2 -23695.108} C_VEL
LIN {X 0,Y 173.324,Z 509.405,A -85,B 0,C 180,E1 -23698.453,E2 -23698.453} C_VEL
LIN {X 0,Y 176.515,Z 501.173,A -85,B 0,C 180,E1 -23701.171,E2 -23701.171} C_VEL
LIN {X 0,Y 179.603,Z 492.129,A -85,B 0,C 180,E1 -23703.553,E2 -23703.553} C_VEL
LIN {X 0,Y 183.033,Z 481.575,A -85,B 0,C 180,E1 -23705.656,E2 -23705.656} C_VEL
LIN {X 0,Y 185.904,Z 470.029,A -85,B 0,C 180,E1 -23707.494,E2 -23707.494} C_VEL
LIN {X 0,Y 188.165,Z 458.718,A -85,B 0,C 180,E1 -23708.847,E2 -23708.847} C_VEL
LIN {X 0,Y 189.703,Z 445.877,A -85,B 0,C 180,E1 -23710.022,E2 -23710.022} C_VEL
LIN {X 0,Y 190.569,Z 433.395,A -85,B 0,C 180,E1 -23710.772,E2 -23710.772} C_VEL
LIN {X 0,Y 191.636,Z 405.693,A -85,B 0,C 180,E1 -23711.879,E2 -23711.879} C_VEL
LIN {X 0,Y 185.991,Z 394.398,A -85,B 0,C 180,E1 -23714.114,E2 -23714.114} C_VEL
LIN {X 0,Y 179.54,Z 383.344,A -85,B 0,C 180,E1 -23716.858,E2 -23716.858} C_VEL
LIN {X 0,Y 173.706,Z 374.56,A -85,B 0,C 180,E1 -23719.583,E2 -23719.583} C_VEL
LIN {X 0,Y 170.838,Z 370.483,A -85,B 0,C 180,E1 -23721.039,E2 -23721.039} C_VEL
LIN {X 0,Y 168.122,Z 366.672,A -85,B 0,C 180,E1 -23722.506,E2 -23722.506} C_VEL
LIN {X 0,Y 165.593,Z 363.186,A -85,B 0,C 180,E1 -23723.961,E2 -23723.961} C_VEL
LIN {X 0,Y 164.371,Z 361.868,A -85,B 0,C 180,E1 -23724.672,E2 -23724.672} C_VEL
LIN {X 0,Y 162.131,Z 358.993,A -85,B 0,C 180,E1 -23726.075,E2 -23726.075} C_VEL
LIN {X 0,Y 161.337,Z 357.483,A -85,B 0,C 180,E1 -23726.636,E2 -23726.636} C_VEL
LIN {X 0,Y 158.707,Z 355.236,A -85,B 0,C 180,E1 -23728.358,E2 -23728.358} C_VEL
LIN {X 0,Y 157.404,Z 352.445,A -85,B 0,C 180,E1 -23729.662,E2 -23729.662} C_VEL
LIN {X 0,Y 157.271,Z 351.925,A -85,B 0,C 180,E1 -23730.557,E2 -23730.557} C_VEL
LIN {X 0,Y 157.308,Z 351.834,A -85,B 0,C 180,E1 -23733.463,E2 -23733.463} C_VEL
LIN {X 0,Y 157.357,Z 351.861,A -85,B 0,C 180,E1 -23739.702,E2 -23739.702} C_VEL
LIN {X 0,Y 157.411,Z 351.853,A -85,B 0,C 180,E1 -23744.461,E2 -23744.461} C_VEL
LIN {X 0,Y 157.683,Z 351.832,A -85,B 0,C 180,E1 -23749.73,E2 -23749.73} C_VEL
LIN {X 0,Y 157.755,Z 351.806,A -85,B 0,C 180,E1 -23752.319,E2 -23752.319} C_VEL
LIN {X 0,Y 158.232,Z 351.747,A -85,B 0,C 180,E1 -23760,E2 -23760} C_VEL
LIN {X 0,Y 157.755,Z 351.812,A -85,B 0,C 180,E1 -23767.68,E2 -23767.68} C_VEL
LIN {X 0,Y 157.63,Z 351.83,A -85,B 0,C 180,E1 -23771.228,E2 -23771.228} C_VEL
LIN {X 0,Y 157.43,Z 351.87,A -85,B 0,C 180,E1 -23775.536,E2 -23775.536} C_VEL
LIN {X 0,Y 157.329,Z 351.836,A -85,B 0,C 180,E1 -23780.938,E2 -23780.938} C_VEL
LIN {X 0,Y 157.347,Z 352.172,A -85,B 0,C 180,E1 -23783.703,E2 -23783.703} C_VEL
LIN {X 0,Y 158.75,Z 356.326,A -85,B 0,C 180,E1 -23787.699,E2 -23787.699} C_VEL
LIN {X 0,Y 160.261,Z 360.466,A -85,B 0,C 180,E1 -23791.016,E2 -23791.016} C_VEL
LIN {X 0,Y 164.198,Z 366.927,A -85,B 0,C 180,E1 -23793.71,E2 -23793.71} C_VEL
LIN {X 0,Y 169.143,Z 375.383,A -85,B 0,C 180,E1 -23796.643,E2 -23796.643} C_VEL
LIN {X 0,Y 172.777,Z 382.184,A -85,B 0,C 180,E1 -23798.619,E2 -23798.619} C_VEL
LIN {X 0,Y 177.515,Z 391.614,A -85,B 0,C 180,E1 -23800.996,E2 -23800.996} C_VEL
LIN {X 0,Y 182.713,Z 403.5,A -85,B 0,C 180,E1 -23803.437,E2 -23803.437} C_VEL
LIN {X 0,Y 185.417,Z 410.731,A -85,B 0,C 180,E1 -23804.669,E2 -23804.669} C_VEL
LIN {X 0,Y 187.375,Z 439.282,A -85,B 0,C 180,E1 -23806.719,E2 -23806.719} C_VEL
LIN {X 0,Y 188.292,Z 462.169,A -85,B 0,C 180,E1 -23808.114,E2 -23808.114} C_VEL
LIN {X 0,Y 187.127,Z 479.642,A -85,B 0,C 180,E1 -23808.814,E2 -23808.814} C_VEL
LIN {X 0,Y 185.41,Z 492.185,A -85,B 0,C 180,E1 -23809.623,E2 -23809.623} C_VEL
LIN {X 0,Y 182.809,Z 504.827,A -85,B 0,C 180,E1 -23810.808,E2 -23810.808} C_VEL
LIN {X 0,Y 179.653,Z 516.554,A -85,B 0,C 180,E1 -23812.321,E2 -23812.321} C_VEL
LIN {X 0,Y 176.005,Z 527.91,A -85,B 0,C 180,E1 -23814.269,E2 -23814.269} C_VEL
LIN {X 0,Y 172.052,Z 538.147,A -85,B 0,C 180,E1 -23816.534,E2 -23816.534} C_VEL
LIN {X 0,Y 168.231,Z 547.419,A -85,B 0,C 180,E1 -23819.22,E2 -23819.22} C_VEL
LIN {X 0,Y 164.235,Z 556.497,A -85,B 0,C 180,E1 -23822.612,E2 -23822.612} C_VEL
LIN {X 0,Y 161.422,Z 562.947,A -85,B 0,C 180,E1 -23825.705,E2 -23825.705} C_VEL
LIN {X 0,Y 158.816,Z 568.859,A -85,B 0,C 180,E1 -23829.267,E2 -23829.267} C_VEL
LIN {X 0,Y 157.68,Z 572.13,A -85,B 0,C 180,E1 -23831.687,E2 -23831.687} C_VEL
LIN {X 0,Y 156.341,Z 574.427,A -85,B 0,C 180,E1 -23833.613,E2 -23833.613} C_VEL
LIN {X 0,Y 152.716,Z 577.376,A -85,B 0,C 180,E1 -23836.859,E2 -23836.859} C_VEL
LIN {X 0,Y 150.033,Z 579.13,A -85,B 0,C 180,E1 -23839.624,E2 -23839.624} C_VEL
LIN {X 0,Y 149.026,Z 580.2,A -85,B 0,C 180,E1 -23841.829,E2 -23841.829} C_VEL
LIN {X 0,Y 149.003,Z 580.52,A -85,B 0,C 180,E1 -23842.58,E2 -23842.58} C_VEL
LIN {X 0,Y 149.759,Z 582.089,A -85,B 0,C 180,E1 -23847.31,E2 -23847.31} C_VEL
LIN {X 0,Y 150.426,Z 582.413,A -85,B 0,C 180,E1 -23850,E2 -23850} C_VEL
LIN {X 0,Y 149.77,Z 582.076,A -85,B 0,C 180,E1 -23852.69,E2 -23852.69} C_VEL
LIN {X 0,Y 149.292,Z 581.332,A -85,B 0,C 180,E1 -23855.402,E2 -23855.402} C_VEL
LIN {X 0,Y 148.953,Z 580.174,A -85,B 0,C 180,E1 -23858.137,E2 -23858.137} C_VEL
LIN {X 0,Y 149.021,Z 577.635,A -85,B 0,C 180,E1 -23862.252,E2 -23862.252} C_VEL
LIN {X 0,Y 149.813,Z 574.108,A -85,B 0,C 180,E1 -23866.348,E2 -23866.348} C_VEL
LIN {X 0,Y 151.422,Z 569.525,A -85,B 0,C 180,E1 -23870.371,E2 -23870.371} C_VEL
LIN {X 0,Y 154.501,Z 562.728,A -85,B 0,C 180,E1 -23874.883,E2 -23874.883} C_VEL
LIN {X 0,Y 157.897,Z 555.325,A -85,B 0,C 180,E1 -23878.586,E2 -23878.586} C_VEL
LIN {X 0,Y 162.138,Z 546.217,A -85,B 0,C 180,E1 -23882.071,E2 -23882.071} C_VEL
LIN {X 0,Y 166.163,Z 536.896,A -85,B 0,C 180,E1 -23884.819,E2 -23884.819} C_VEL
LIN {X 0,Y 170.282,Z 526.583,A -85,B 0,C 180,E1 -23887.128,E2 -23887.128} C_VEL
LIN {X 0,Y 174.127,Z 515.159,A -85,B 0,C 180,E1 -23889.097,E2 -23889.097} C_VEL
LIN {X 0,Y 177.346,Z 503.303,A -85,B 0,C 180,E1 -23890.646,E2 -23890.646} C_VEL
LIN {X 0,Y 179.954,Z 490.768,A -85,B 0,C 180,E1 -23891.822,E2 -23891.822} C_VEL
LIN {X 0,Y 181.863,Z 476.976,A -85,B 0,C 180,E1 -23892.69,E2 -23892.69} C_VEL
LIN {X 0,Y 182.831,Z 461.944,A -85,B 0,C 180,E1 -23893.297,E2 -23893.297} C_VEL
LIN {X 0,Y 181.688,Z 434.14,A -85,B 0,C 180,E1 -23895.107,E2 -23895.107} C_VEL
LIN {X 0,Y 180.26,Z 412.702,A -85,B 0,C 180,E1 -23896.734,E2 -23896.734} C_VEL
LIN {X 0,Y 174.942,Z 399.556,A -85,B 0,C 180,E1 -23899.34,E2 -23899.34} C_VEL
LIN {X 0,Y 170.04,Z 389.098,A -85,B 0,C 180,E1 -23901.913,E2 -23901.913} C_VEL
LIN {X 0,Y 166.776,Z 382.771,A -85,B 0,C 180,E1 -23903.754,E2 -23903.754} C_VEL
LIN {X 0,Y 164.358,Z 378.209,A -85,B 0,C 180,E1 -23905.209,E2 -23905.209} C_VEL
LIN {X 0,Y 160.842,Z 372.051,A -85,B 0,C 180,E1 -23907.469,E2 -23907.469} C_VEL
LIN {X 0,Y 156.581,Z 365.09,A -85,B 0,C 180,E1 -23910.511,E2 -23910.511} C_VEL
LIN {X 0,Y 152.627,Z 359.013,A -85,B 0,C 180,E1 -23913.784,E2 -23913.784} C_VEL
LIN {X 0,Y 151.941,Z 357.647,A -85,B 0,C 180,E1 -23914.668,E2 -23914.668} C_VEL
LIN {X 0,Y 150.368,Z 352.854,A -85,B 0,C 180,E1 -23919.778,E2 -23919.778} C_VEL
LIN {X 0,Y 150.349,Z 352.758,A -85,B 0,C 180,E1 -23923.712,E2 -23923.712} C_VEL
LIN {X 0,Y 150.606,Z 352.712,A -85,B 0,C 180,E1 -23929.242,E2 -23929.242} C_VEL
LIN {X 0,Y 150.696,Z 352.695,A -85,B 0,C 180,E1 -23931.957,E2 -23931.957} C_VEL
LIN {X 0,Y 151.193,Z 352.624,A -85,B 0,C 180,E1 -23940,E2 -23940} C_VEL
LIN {X 0,Y 150.678,Z 352.686,A -85,B 0,C 180,E1 -23948.044,E2 -23948.044} C_VEL
LIN {X 0,Y 150.571,Z 352.727,A -85,B 0,C 180,E1 -23951.43,E2 -23951.43} C_VEL
LIN {X 0,Y 150.32,Z 352.741,A -85,B 0,C 180,E1 -23956.292,E2 -23956.292} C_VEL
LIN {X 0,Y 150.281,Z 352.741,A -85,B 0,C 180,E1 -23960.724,E2 -23960.724} C_VEL
LIN {X 0,Y 150.25,Z 353.059,A -85,B 0,C 180,E1 -23965.222,E2 -23965.222} C_VEL
LIN {X 0,Y 150.583,Z 354.128,A -85,B 0,C 180,E1 -23966.14,E2 -23966.14} C_VEL
LIN {X 0,Y 152.111,Z 356.758,A -85,B 0,C 180,E1 -23967.652,E2 -23967.652} C_VEL
LIN {X 0,Y 154.817,Z 358.728,A -85,B 0,C 180,E1 -23969.77,E2 -23969.77} C_VEL
LIN {X 0,Y 156.636,Z 361.921,A -85,B 0,C 180,E1 -23971.245,E2 -23971.245} C_VEL
LIN {X 0,Y 158.989,Z 364.202,A -85,B 0,C 180,E1 -23972.861,E2 -23972.861} C_VEL
LIN {X 0,Y 161.391,Z 367.625,A -85,B 0,C 180,E1 -23974.479,E2 -23974.479} C_VEL
LIN {X 0,Y 162.718,Z 369.166,A -85,B 0,C 180,E1 -23975.298,E2 -23975.298} C_VEL
LIN {X 0,Y 166.848,Z 374.988,A -85,B 0,C 180,E1 -23977.737,E2 -23977.737} C_VEL
LIN {X 0,Y 171.85,Z 382.246,A -85,B 0,C 180,E1 -23980.387,E2 -23980.387} C_VEL
LIN {X 0,Y 177.867,Z 391.973,A -85,B 0,C 180,E1 -23983.268,E2 -23983.268} C_VEL
LIN {X 0,Y 183.982,Z 403.343,A -85,B 0,C 180,E1 -23985.942,E2 -23985.942} C_VEL
LIN {X 0,Y 186.277,Z 408.143,A -85,B 0,C 180,E1 -23986.898,E2 -23986.898} C_VEL
LIN {X 0,Y 184.859,Z 439.367,A -85,B 0,C 180,E1 -23988.22,E2 -23988.22} C_VEL
LIN {X 0,Y 183.491,Z 452.668,A -85,B 0,C 180,E1 -23989.19,E2 -23989.19} C_VEL
LIN {X 0,Y 181.511,Z 464.95,A -85,B 0,C 180,E1 -23990.493,E2 -23990.493} C_VEL
LIN {X 0,Y 178.952,Z 476.291,A -85,B 0,C 180,E1 -23992.099,E2 -23992.099} C_VEL
LIN {X 0,Y 175.921,Z 486.461,A -85,B 0,C 180,E1 -23993.896,E2 -23993.896} C_VEL
LIN {X 0,Y 172.706,Z 495.736,A -85,B 0,C 180,E1 -23995.977,E2 -23995.977} C_VEL
LIN {X 0,Y 169.171,Z 505.178,A -85,B 0,C 180,E1 -23998.715,E2 -23998.715} C_VEL
LIN {X 0,Y 165.83,Z 512.912,A -85,B 0,C 180,E1 -24001.525,E2 -24001.525} C_VEL
LIN {X 0,Y 162.202,Z 520.565,A -85,B 0,C 180,E1 -24005.079,E2 -24005.079} C_VEL
LIN {X 0,Y 158.712,Z 527.364,A -85,B 0,C 180,E1 -24009.253,E2 -24009.253} C_VEL
LIN {X 0,Y 156.124,Z 531.969,A -85,B 0,C 180,E1 -24012.987,E2 -24012.987} C_VEL
LIN {X 0,Y 153.883,Z 535.515,A -85,B 0,C 180,E1 -24016.8,E2 -24016.8} C_VEL
LIN {X 0,Y 152.768,Z 537.337,A -85,B 0,C 180,E1 -24019.396,E2 -24019.396} C_VEL
LIN {X 0,Y 152.168,Z 538.667,A -85,B 0,C 180,E1 -24022.036,E2 -24022.036} C_VEL
LIN {X 0,Y 151.352,Z 540.212,A -85,B 0,C 180,E1 -24027.339,E2 -24027.339} C_VEL
LIN {X 0,Y 151.248,Z 540.433,A -85,B 0,C 180,E1 -24030,E2 -24030} C_VEL
LIN {X 0,Y 151.352,Z 540.243,A -85,B 0,C 180,E1 -24032.661,E2 -24032.661} C_VEL
LIN {X 0,Y 152.161,Z 538.737,A -85,B 0,C 180,E1 -24037.965,E2 -24037.965} C_VEL
LIN {X 0,Y 152.75,Z 537.44,A -85,B 0,C 180,E1 -24040.605,E2 -24040.605} C_VEL
LIN {X 0,Y 154.659,Z 534.595,A -85,B 0,C 180,E1 -24044.473,E2 -24044.473} C_VEL
LIN {X 0,Y 156.987,Z 530.76,A -85,B 0,C 180,E1 -24048.262,E2 -24048.262} C_VEL
LIN {X 0,Y 159.665,Z 525.67,A -85,B 0,C 180,E1 -24052.106,E2 -24052.106} C_VEL
LIN {X 0,Y 163.431,Z 518.418,A -85,B 0,C 180,E1 -24056.153,E2 -24056.153} C_VEL
LIN {X 0,Y 167.178,Z 510.381,A -85,B 0,C 180,E1 -24059.601,E2 -24059.601} C_VEL
LIN {X 0,Y 170.538,Z 502.148,A -85,B 0,C 180,E1 -24062.393,E2 -24062.393} C_VEL
LIN {X 0,Y 173.795,Z 493.102,A -85,B 0,C 180,E1 -24064.833,E2 -24064.833} C_VEL
LIN {X 0,Y 177.372,Z 482.547,A -85,B 0,C 180,E1 -24066.979,E2 -24066.979} C_VEL
LIN {X 0,Y 180.378,Z 471.002,A -85,B 0,C 180,E1 -24068.853,E2 -24068.853} C_VEL
LIN {X 0,Y 182.742,Z 459.689,A -85,B 0,C 180,E1 -24070.23,E2 -24070.23} C_VEL
LIN {X 0,Y 184.391,Z 446.602,A -85,B 0,C 180,E1 -24071.447,E2 -24071.447} C_VEL
LIN {X 0,Y 185.292,Z 434.789,A -85,B 0,C 180,E1 -24072.167,E2 -24072.167} C_VEL
LIN {X 0,Y 186.437,Z 408.376,A -85,B 0,C 180,E1 -24073.237,E2 -24073.237} C_VEL
LIN {X 0,Y 181.02,Z 397.474,A -85,B 0,C 180,E1 -24075.54,E2 -24075.54} C_VEL
LIN {X 0,Y 174.589,Z 386.493,A -85,B 0,C 180,E1 -24078.488,E2 -24078.488} C_VEL
LIN {X 0,Y 168.21,Z 376.738,A -85,B 0,C 180,E1 -24081.765,E2 -24081.765} C_VEL
LIN {X 0,Y 164.783,Z 372.066,A -85,B 0,C 180,E1 -24083.703,E2 -24083.703} C_VEL
LIN {X 0,Y 161.951,Z 368.174,A -85,B 0,C 180,E1 -24085.446,E2 -24085.446} C_VEL
LIN {X 0,Y 159.393,Z 364.904,A -85,B 0,C 180,E1 -24087.129,E2 -24087.129} C_VEL
LIN {X 0,Y 158.603,Z 363.635,A -85,B 0,C 180,E1 -24087.698,E2 -24087.698} C_VEL
LIN {X 0,Y 155.961,Z 360.884,A -85,B 0,C 180,E1 -24089.581,E2 -24089.581} C_VEL
LIN {X 0,Y 154.566,Z 358.487,A -85,B 0,C 180,E1 -24090.738,E2 -24090.738} C_VEL
LIN {X 0,Y 151.994,Z 356.618,A -85,B 0,C 180,E1 -24092.79,E2 -24092.79} C_VEL
LIN {X 0,Y 150.368,Z 353.52,A -85,B 0,C 180,E1 -24094.603,E2 -24094.603} C_VEL
LIN {X 0,Y 150.247,Z 352.804,A -85,B 0,C 180,E1 -24095.839,E2 -24095.839} C_VEL
LIN {X 0,Y 150.298,Z 352.748,A -85,B 0,C 180,E1 -24100.893,E2 -24100.893} C_VEL
LIN {X 0,Y 150.405,Z 352.725,A -85,B 0,C 180,E1 -24106.489,E2 -24106.489} C_VEL
LIN {X 0,Y 150.603,Z 352.721,A -85,B 0,C 180,E1 -24109.242,E2 -24109.242} C_VEL
LIN {X 0,Y 150.678,Z 352.687,A -85,B 0,C 180,E1 -24111.956,E2 -24111.956} C_VEL
LIN {X 0,Y 151.193,Z 352.624,A -85,B 0,C 180,E1 -24120,E2 -24120} C_VEL
LIN {X 0,Y 150.678,Z 352.697,A -85,B 0,C 180,E1 -24128.044,E2 -24128.044} C_VEL
LIN {X 0,Y 150.572,Z 352.707,A -85,B 0,C 180,E1 -24131.431,E2 -24131.431} C_VEL
LIN {X 0,Y 150.342,Z 352.758,A -85,B 0,C 180,E1 -24136.289,E2 -24136.289} C_VEL
LIN {X 0,Y 150.368,Z 352.907,A -85,B 0,C 180,E1 -24140.093,E2 -24140.093} C_VEL
LIN {X 0,Y 151.858,Z 357.473,A -85,B 0,C 180,E1 -24144.98,E2 -24144.98} C_VEL
LIN {X 0,Y 153.481,Z 360.553,A -85,B 0,C 180,E1 -24146.792,E2 -24146.792} C_VEL
LIN {X 0,Y 157.764,Z 366.892,A -85,B 0,C 180,E1 -24150.169,E2 -24150.169} C_VEL
LIN {X 0,Y 162.236,Z 374.388,A -85,B 0,C 180,E1 -24153.275,E2 -24153.275} C_VEL
LIN {X 0,Y 165.869,Z 380.837,A -85,B 0,C 180,E1 -24155.54,E2 -24155.54} C_VEL
LIN {X 0,Y 169.28,Z 387.476,A -85,B 0,C 180,E1 -24157.519,E2 -24157.519} C_VEL
LIN {X 0,Y 173.748,Z 396.751,A -85,B 0,C 180,E1 -24159.914,E2 -24159.914} C_VEL
LIN {X 0,Y 178.486,Z 407.896,A -85,B 0,C 180,E1 -24162.287,E2 -24162.287} C_VEL
LIN {X 0,Y 180.472,Z 413.141,A -85,B 0,C 180,E1 -24163.247,E2 -24163.247} C_VEL
LIN {X 0,Y 182.285,Z 443.398,A -85,B 0,C 180,E1 -24165.464,E2 -24165.464} C_VEL
LIN {X 0,Y 182.946,Z 463.276,A -85,B 0,C 180,E1 -24166.703,E2 -24166.703} C_VEL
LIN {X 0,Y 181.693,Z 479.862,A -85,B 0,C 180,E1 -24167.396,E2 -24167.396} C_VEL
LIN {X 0,Y 180.01,Z 491.41,A -85,B 0,C 180,E1 -24168.17,E2 -24168.17} C_VEL
LIN {X 0,Y 177.368,Z 503.846,A -85,B 0,C 180,E1 -24169.36,E2 -24169.36} C_VEL
LIN {X 0,Y 174.075,Z 515.568,A -85,B 0,C 180,E1 -24170.889,E2 -24170.889} C_VEL
LIN {X 0,Y 170.289,Z 526.925,A -85,B 0,C 180,E1 -24172.873,E2 -24172.873} C_VEL
LIN {X 0,Y 166.165,Z 537.16,A -85,B 0,C 180,E1 -24175.182,E2 -24175.182} C_VEL
LIN {X 0,Y 162.13,Z 546.427,A -85,B 0,C 180,E1 -24177.927,E2 -24177.927} C_VEL
LIN {X 0,Y 157.916,Z 555.503,A -85,B 0,C 180,E1 -24181.418,E2 -24181.418} C_VEL
LIN {X 0,Y 154.511,Z 562.868,A -85,B 0,C 180,E1 -24185.119,E2 -24185.119} C_VEL
LIN {X 0,Y 151.405,Z 569.627,A -85,B 0,C 180,E1 -24189.627,E2 -24189.627} C_VEL
LIN {X 0,Y 149.822,Z 574.188,A -85,B 0,C 180,E1 -24193.653,E2 -24193.653} C_VEL
LIN {X 0,Y 149.022,Z 577.687,A -85,B 0,C 180,E1 -24197.747,E2 -24197.747} C_VEL
LIN {X 0,Y 149.003,Z 580.52,A -85,B 0,C 180,E1 -24202.58,E2 -24202.58} C_VEL
LIN {X 0,Y 148.56,Z 581.354,A -85,B 0,C 180,E1 -24204.835,E2 -24204.835} C_VEL
LIN {X 0,Y 147.199,Z 581.711,A -85,B 0,C 180,E1 -24207.082,E2 -24207.082} C_VEL
LIN {X 0,Y 143.666,Z 581.373,A -85,B 0,C 180,E1 -24211.661,E2 -24211.661} C_VEL
LIN {X 0,Y 142.281,Z 580.55,A -85,B 0,C 180,E1 -24214.862,E2 -24214.862} C_VEL
LIN {X 0,Y 141.864,Z 579.177,A -85,B 0,C 180,E1 -24218.547,E2 -24218.547} C_VEL
LIN {X 0,Y 142.017,Z 576.636,A -85,B 0,C 180,E1 -24222.867,E2 -24222.867} C_VEL
LIN {X 0,Y 142.94,Z 573.109,A -85,B 0,C 180,E1 -24227.158,E2 -24227.158} C_VEL
LIN {X 0,Y 144.722,Z 568.527,A -85,B 0,C 180,E1 -24231.359,E2 -24231.359} C_VEL
LIN {X 0,Y 147.521,Z 562.797,A -85,B 0,C 180,E1 -24235.389,E2 -24235.389} C_VEL
LIN {X 0,Y 151.011,Z 555.694,A -85,B 0,C 180,E1 -24239.252,E2 -24239.252} C_VEL
LIN {X 0,Y 155.362,Z 546.879,A -85,B 0,C 180,E1 -24242.876,E2 -24242.876} C_VEL
LIN {X 0,Y 159.482,Z 537.885,A -85,B 0,C 180,E1 -24245.724,E2 -24245.724} C_VEL
LIN {X 0,Y 163.691,Z 528.068,A -85,B 0,C 180,E1 -24248.11,E2 -24248.11} C_VEL
LIN {X 0,Y 167.672,Z 517.333,A -85,B 0,C 180,E1 -24250.123,E2 -24250.123} C_VEL
LIN {X 0,Y 171.214,Z 505.306,A -85,B 0,C 180,E1 -24251.837,E2 -24251.837} C_VEL
LIN {X 0,Y 174.143,Z 492.816,A -85,B 0,C 180,E1 -24253.121,E2 -24253.121} C_VEL
LIN {X 0,Y 176.24,Z 480.094,A -85,B 0,C 180,E1 -24254.037,E2 -24254.037} C_VEL
LIN {X 0,Y 177.458,Z 466.901,A -85,B 0,C 180,E1 -24254.624,E2 -24254.624} C_VEL
LIN {X 0,Y 177.541,Z 459.407,A -85,B 0,C 180,E1 -24255.01,E2 -24255.01} C_VEL
LIN {X 0,Y 176.262,Z 428.692,A -85,B 0,C 180,E1 -24257.155,E2 -24257.155} C_VEL
LIN {X 0,Y 175.402,Z 415.511,A -85,B 0,C 180,E1 -24258.221,E2 -24258.221} C_VEL
LIN {X 0,Y 170.917,Z 404.017,A -85,B 0,C 180,E1 -24260.596,E2 -24260.596} C_VEL
LIN {X 0,Y 166.446,Z 394.122,A -85,B 0,C 180,E1 -24263.115,E2 -24263.115} C_VEL
LIN {X 0,Y 162.706,Z 386.556,A -85,B 0,C 180,E1 -24265.399,E2 -24265.399} C_VEL
LIN {X 0,Y 160.389,Z 382.263,A -85,B 0,C 180,E1 -24266.907,E2 -24266.907} C_VEL
LIN {X 0,Y 157.792,Z 377.471,A -85,B 0,C 180,E1 -24268.724,E2 -24268.724} C_VEL
LIN {X 0,Y 153.987,Z 370.991,A -85,B 0,C 180,E1 -24271.638,E2 -24271.638} C_VEL
LIN {X 0,Y 150.083,Z 364.696,A -85,B 0,C 180,E1 -24275.074,E2 -24275.074} C_VEL
LIN {X 0,Y 144.886,Z 357.267,A -85,B 0,C 180,E1 -24280.704,E2 -24280.704} C_VEL
LIN {X 0,Y 143.43,Z 354.399,A -85,B 0,C 180,E1 -24283.27,E2 -24283.27} C_VEL
LIN {X 0,Y 143.324,Z 353.705,A -85,B 0,C 180,E1 -24284.718,E2 -24284.718} C_VEL
LIN {X 0,Y 143.532,Z 353.586,A -85,B 0,C 180,E1 -24288.705,E2 -24288.705} C_VEL
LIN {X 0,Y 143.618,Z 353.58,A -85,B 0,C 180,E1 -24291.558,E2 -24291.558} C_VEL
LIN {X 0,Y 144.152,Z 353.5,A -85,B 0,C 180,E1 -24300,E2 -24300} C_VEL
LIN {X 0,Y 143.604,Z 353.567,A -85,B 0,C 180,E1 -24308.443,E2 -24308.443} C_VEL
LIN {X 0,Y 143.497,Z 353.604,A -85,B 0,C 180,E1 -24311.618,E2 -24311.618} C_VEL
LIN {X 0,Y 143.268,Z 353.924,A -85,B 0,C 180,E1 -24318.131,E2 -24318.131} C_VEL
LIN {X 0,Y 143.551,Z 354.954,A -85,B 0,C 180,E1 -24319.39,E2 -24319.39} C_VEL
LIN {X 0,Y 145.176,Z 357.737,A -85,B 0,C 180,E1 -24321.672,E2 -24321.672} C_VEL
LIN {X 0,Y 148.169,Z 359.876,A -85,B 0,C 180,E1 -24324.802,E2 -24324.802} C_VEL
LIN {X 0,Y 149.961,Z 363.008,A -85,B 0,C 180,E1 -24326.651,E2 -24326.651} C_VEL
LIN {X 0,Y 152.643,Z 365.417,A -85,B 0,C 180,E1 -24328.912,E2 -24328.912} C_VEL
LIN {X 0,Y 154.853,Z 368.734,A -85,B 0,C 180,E1 -24330.723,E2 -24330.723} C_VEL
LIN {X 0,Y 156.595,Z 370.609,A -85,B 0,C 180,E1 -24331.986,E2 -24331.986} C_VEL
LIN {X 0,Y 159.281,Z 374.198,A -85,B 0,C 180,E1 -24333.853,E2 -24333.853} C_VEL
LIN {X 0,Y 164.054,Z 381.012,A -85,B 0,C 180,E1 -24336.853,E2 -24336.853} C_VEL
LIN {X 0,Y 169.976,Z 390.012,A -85,B 0,C 180,E1 -24340.124,E2 -24340.124} C_VEL
LIN {X 0,Y 175.71,Z 399.97,A -85,B 0,C 180,E1 -24342.969,E2 -24342.969} C_VEL
LIN {X 0,Y 181.137,Z 410.751,A -85,B 0,C 180,E1 -24345.445,E2 -24345.445} C_VEL
LIN {X 0,Y 179.679,Z 440.359,A -85,B 0,C 180,E1 -24346.726,E2 -24346.726} C_VEL
LIN {X 0,Y 178.273,Z 453.325,A -85,B 0,C 180,E1 -24347.684,E2 -24347.684} C_VEL
LIN {X 0,Y 176.145,Z 465.935,A -85,B 0,C 180,E1 -24349.038,E2 -24349.038} C_VEL
LIN {X 0,Y 173.204,Z 478.249,A -85,B 0,C 180,E1 -24350.838,E2 -24350.838} C_VEL
LIN {X 0,Y 169.873,Z 488.714,A -85,B 0,C 180,E1 -24352.767,E2 -24352.767} C_VEL
LIN {X 0,Y 166.564,Z 497.762,A -85,B 0,C 180,E1 -24354.909,E2 -24354.909} C_VEL
LIN {X 0,Y 163.204,Z 506.159,A -85,B 0,C 180,E1 -24357.434,E2 -24357.434} C_VEL
LIN {X 0,Y 159.687,Z 513.892,A -85,B 0,C 180,E1 -24360.323,E2 -24360.323} C_VEL
LIN {X 0,Y 155.856,Z 521.545,A -85,B 0,C 180,E1 -24363.991,E2 -24363.991} C_VEL
LIN {X 0,Y 152.161,Z 528.343,A -85,B 0,C 180,E1 -24368.315,E2 -24368.315} C_VEL
LIN {X 0,Y 149.418,Z 532.948,A -85,B 0,C 180,E1 -24372.198,E2 -24372.198} C_VEL
LIN {X 0,Y 147.047,Z 536.494,A -85,B 0,C 180,E1 -24376.174,E2 -24376.174} C_VEL
LIN {X 0,Y 145.862,Z 538.316,A -85,B 0,C 180,E1 -24378.888,E2 -24378.888} C_VEL
LIN {X 0,Y 145.21,Z 539.645,A -85,B 0,C 180,E1 -24381.652,E2 -24381.652} C_VEL
LIN {X 0,Y 144.332,Z 541.19,A -85,B 0,C 180,E1 -24387.209,E2 -24387.209} C_VEL
LIN {X 0,Y 144.221,Z 541.411,A -85,B 0,C 180,E1 -24390,E2 -24390} C_VEL
LIN {X 0,Y 144.331,Z 541.22,A -85,B 0,C 180,E1 -24392.791,E2 -24392.791} C_VEL
LIN {X 0,Y 145.202,Z 539.715,A -85,B 0,C 180,E1 -24398.349,E2 -24398.349} C_VEL
LIN {X 0,Y 145.844,Z 538.417,A -85,B 0,C 180,E1 -24401.113,E2 -24401.113} C_VEL
LIN {X 0,Y 147.864,Z 535.572,A -85,B 0,C 180,E1 -24405.154,E2 -24405.154} C_VEL
LIN {X 0,Y 150.329,Z 531.737,A -85,B 0,C 180,E1 -24409.102,E2 -24409.102} C_VEL
LIN {X 0,Y 153.177,Z 526.646,A -85,B 0,C 180,E1 -24413.096,E2 -24413.096} C_VEL
LIN {X 0,Y 157.153,Z 519.394,A -85,B 0,C 180,E1 -24417.283,E2 -24417.283} C_VEL
LIN {X 0,Y 161.104,Z 511.357,A -85,B 0,C 180,E1 -24420.835,E2 -24420.835} C_VEL
LIN {X 0,Y 164.645,Z 503.123,A -85,B 0,C 180,E1 -24423.704,E2 -24423.704} C_VEL
LIN {X 0,Y 168.08,Z 494.076,A -85,B 0,C 180,E1 -24426.2,E2 -24426.2} C_VEL
LIN {X 0,Y 171.811,Z 483.52,A -85,B 0,C 180,E1 -24428.388,E2 -24428.388} C_VEL
LIN {X 0,Y 174.961,Z 471.974,A -85,B 0,C 180,E1 -24430.297,E2 -24430.297} C_VEL
LIN {X 0,Y 177.43,Z 460.66,A -85,B 0,C 180,E1 -24431.697,E2 -24431.697} C_VEL
LIN {X 0,Y 179.087,Z 448.489,A -85,B 0,C 180,E1 -24432.866,E2 -24432.866} C_VEL
LIN {X 0,Y 180.137,Z 436.059,A -85,B 0,C 180,E1 -24433.65,E2 -24433.65} C_VEL
LIN {X 0,Y 181.189,Z 410.748,A -85,B 0,C 180,E1 -24434.741,E2 -24434.741} C_VEL
LIN {X 0,Y 176.476,Z 401.246,A -85,B 0,C 180,E1 -24436.893,E2 -24436.893} C_VEL
LIN {X 0,Y 171.06,Z 391.761,A -85,B 0,C 180,E1 -24439.547,E2 -24439.547} C_VEL
LIN {X 0,Y 165.154,Z 382.474,A -85,B 0,C 180,E1 -24442.766,E2 -24442.766} C_VEL
LIN {X 0,Y 161.696,Z 377.614,A -85,B 0,C 180,E1 -24444.845,E2 -24444.845} C_VEL
LIN {X 0,Y 159.034,Z 373.905,A -85,B 0,C 180,E1 -24446.587,E2 -24446.587} C_VEL
LIN {X 0,Y 156.401,Z 370.181,A -85,B 0,C 180,E1 -24448.465,E2 -24448.465} C_VEL
LIN {X 0,Y 153.309,Z 366.583,A -85,B 0,C 180,E1 -24450.828,E2 -24450.828} C_VEL
LIN {X 0,Y 152.237,Z 364.9,A -85,B 0,C 180,E1 -24451.758,E2 -24451.758} C_VEL
LIN {X 0,Y 149.814,Z 362.776,A -85,B 0,C 180,E1 -24453.846,E2 -24453.846} C_VEL
LIN {X 0,Y 147.951,Z 359.537,A -85,B 0,C 180,E1 -24455.813,E2 -24455.813} C_VEL
LIN {X 0,Y 145.193,Z 357.74,A -85,B 0,C 180,E1 -24458.746,E2 -24458.746} C_VEL
LIN {X 0,Y 143.654,Z 355.255,A -85,B 0,C 180,E1 -24460.903,E2 -24460.903} C_VEL
LIN {X 0,Y 143.293,Z 354.025,A -85,B 0,C 180,E1 -24462.149,E2 -24462.149} C_VEL
LIN {X 0,Y 143.289,Z 353.629,A -85,B 0,C 180,E1 -24464.35,E2 -24464.35} C_VEL
LIN {X 0,Y 143.53,Z 353.607,A -85,B 0,C 180,E1 -24468.705,E2 -24468.705} C_VEL
LIN {X 0,Y 143.604,Z 353.569,A -85,B 0,C 180,E1 -24471.557,E2 -24471.557} C_VEL
LIN {X 0,Y 144.152,Z 353.5,A -85,B 0,C 180,E1 -24480,E2 -24480} C_VEL
LIN {X 0,Y 143.604,Z 353.581,A -85,B 0,C 180,E1 -24488.443,E2 -24488.443} C_VEL
LIN {X 0,Y 143.498,Z 353.586,A -85,B 0,C 180,E1 -24491.62,E2 -24491.62} C_VEL
LIN {X 0,Y 143.348,Z 353.908,A -85,B 0,C 180,E1 -24495.643,E2 -24495.643} C_VEL
LIN {X 0,Y 143.652,Z 355.157,A -85,B 0,C 180,E1 -24497.07,E2 -24497.07} C_VEL
LIN {X 0,Y 146.085,Z 359.056,A -85,B 0,C 180,E1 -24500.442,E2 -24500.442} C_VEL
LIN {X 0,Y 150.311,Z 365.044,A -85,B 0,C 180,E1 -24504.886,E2 -24504.886} C_VEL
LIN {X 0,Y 155.053,Z 372.633,A -85,B 0,C 180,E1 -24508.993,E2 -24508.993} C_VEL
LIN {X 0,Y 159.398,Z 380.265,A -85,B 0,C 180,E1 -24512.222,E2 -24512.222} C_VEL
LIN {X 0,Y 162.724,Z 386.464,A -85,B 0,C 180,E1 -24514.438,E2 -24514.438} C_VEL
LIN {X 0,Y 165.648,Z 392.327,A -85,B 0,C 180,E1 -24516.251,E2 -24516.251} C_VEL
LIN {X 0,Y 169.841,Z 401.323,A -85,B 0,C 180,E1 -24518.665,E2 -24518.665} C_VEL
LIN {X 0,Y 174.67,Z 413.19,A -85,B 0,C 180,E1 -24521.257,E2 -24521.257} C_VEL
LIN {X 0,Y 175.711,Z 416.456,A -85,B 0,C 180,E1 -24521.823,E2 -24521.823} C_VEL
LIN {X 0,Y 177.303,Z 447.008,A -85,B 0,C 180,E1 -24524.115,E2 -24524.115} C_VEL
LIN {X 0,Y 177.738,Z 463.89,A -85,B 0,C 180,E1 -24525.188,E2 -24525.188} C_VEL
LIN {X 0,Y 176.498,Z 479.165,A -85,B 0,C 180,E1 -24525.849,E2 -24525.849} C_VEL
LIN {X 0,Y 174.418,Z 492.237,A -85,B 0,C 180,E1 -24526.766,E2 -24526.766} C_VEL
LIN {X 0,Y 171.765,Z 503.86,A -85,B 0,C 180,E1 -24527.933,E2 -24527.933} C_VEL
LIN {X 0,Y 168.098,Z 516.174,A -85,B 0,C 180,E1 -24529.607,E2 -24529.607} C_VEL
LIN {X 0,Y 164.187,Z 527.202,A -85,B 0,C 180,E1 -24531.636,E2 -24531.636} C_VEL
LIN {X 0,Y 160.386,Z 536.175,A -85,B 0,C 180,E1 -24533.733,E2 -24533.733} C_VEL
LIN {X 0,Y 156.131,Z 545.437,A -85,B 0,C 180,E1 -24536.536,E2 -24536.536} C_VEL
LIN {X 0,Y 151.691,Z 554.513,A -85,B 0,C 180,E1 -24540.129,E2 -24540.129} C_VEL
LIN {X 0,Y 148.045,Z 561.874,A -85,B 0,C 180,E1 -24543.953,E2 -24543.953} C_VEL
LIN {X 0,Y 145.507,Z 566.868,A -85,B 0,C 180,E1 -24547.27,E2 -24547.27} C_VEL
LIN {X 0,Y 143.479,Z 571.809,A -85,B 0,C 180,E1 -24551.435,E2 -24551.435} C_VEL
LIN {X 0,Y 142.247,Z 575.643,A -85,B 0,C 180,E1 -24555.698,E2 -24555.698} C_VEL
LIN {X 0,Y 141.877,Z 577.658,A -85,B 0,C 180,E1 -24558.572,E2 -24558.572} C_VEL
LIN {X 0,Y 142.166,Z 580.359,A -85,B 0,C 180,E1 -24564.326,E2 -24564.326} C_VEL
LIN {X 0,Y 142.675,Z 581.102,A -85,B 0,C 180,E1 -24567.177,E2 -24567.177} C_VEL
LIN {X 0,Y 143.341,Z 581.427,A -85,B 0,C 180,E1 -24570,E2 -24570} C_VEL
LIN {X 0,Y 142.281,Z 580.55,A -85,B 0,C 180,E1 -24574.862,E2 -24574.862} C_VEL
LIN {X 0,Y 141.76,Z 580.046,A -85,B 0,C 180,E1 -24576.424,E2 -24576.424} C_VEL
LIN {X 0,Y 139.619,Z 578.573,A -85,B 0,C 180,E1 -24579.471,E2 -24579.471} C_VEL
LIN {X 0,Y 136.223,Z 575.443,A -85,B 0,C 180,E1 -24584.06,E2 -24584.06} C_VEL
LIN {X 0,Y 135.684,Z 573.531,A -85,B 0,C 180,E1 -24586.421,E2 -24586.421} C_VEL
LIN {X 0,Y 135.826,Z 572.853,A -85,B 0,C 180,E1 -24587.205,E2 -24587.205} C_VEL
LIN {X 0,Y 138.074,Z 567.528,A -85,B 0,C 180,E1 -24592.442,E2 -24592.442} C_VEL
LIN {X 0,Y 141.657,Z 560.735,A -85,B 0,C 180,E1 -24597.317,E2 -24597.317} C_VEL
LIN {X 0,Y 145.493,Z 553.329,A -85,B 0,C 180,E1 -24601.283,E2 -24601.283} C_VEL
LIN {X 0,Y 150.235,Z 544.226,A -85,B 0,C 180,E1 -24604.963,E2 -24604.963} C_VEL
LIN {X 0,Y 154.722,Z 534.914,A -85,B 0,C 180,E1 -24607.821,E2 -24607.821} C_VEL
LIN {X 0,Y 159.198,Z 524.6,A -85,B 0,C 180,E1 -24610.213,E2 -24610.213} C_VEL
LIN {X 0,Y 163.297,Z 513.163,A -85,B 0,C 180,E1 -24612.257,E2 -24612.257} C_VEL
LIN {X 0,Y 166.829,Z 501.315,A -85,B 0,C 180,E1 -24613.824,E2 -24613.824} C_VEL
LIN {X 0,Y 169.651,Z 488.495,A -85,B 0,C 180,E1 -24615.054,E2 -24615.054} C_VEL
LIN {X 0,Y 171.585,Z 475.341,A -85,B 0,C 180,E1 -24615.908,E2 -24615.908} C_VEL
LIN {X 0,Y 172.533,Z 463.608,A -85,B 0,C 180,E1 -24616.394,E2 -24616.394} C_VEL
LIN {X 0,Y 171.668,Z 436.275,A -85,B 0,C 180,E1 -24618.315,E2 -24618.315} C_VEL
LIN {X 0,Y 170.712,Z 418.368,A -85,B 0,C 180,E1 -24619.772,E2 -24619.772} C_VEL
LIN {X 0,Y 166.326,Z 406.89,A -85,B 0,C 180,E1 -24622.296,E2 -24622.296} C_VEL
LIN {X 0,Y 162.223,Z 397.617,A -85,B 0,C 180,E1 -24624.818,E2 -24624.818} C_VEL
LIN {X 0,Y 158.227,Z 389.25,A -85,B 0,C 180,E1 -24627.514,E2 -24627.514} C_VEL
LIN {X 0,Y 154.701,Z 382.71,A -85,B 0,C 180,E1 -24630.117,E2 -24630.117} C_VEL
LIN {X 0,Y 151.355,Z 376.677,A -85,B 0,C 180,E1 -24632.894,E2 -24632.894} C_VEL
LIN {X 0,Y 147.758,Z 370.577,A -85,B 0,C 180,E1 -24636.316,E2 -24636.316} C_VEL
LIN {X 0,Y 143.105,Z 363.634,A -85,B 0,C 180,E1 -24641.755,E2 -24641.755} C_VEL
LIN {X 0,Y 141.304,Z 360.594,A -85,B 0,C 180,E1 -24644.494,E2 -24644.494} C_VEL
LIN {X 0,Y 137.968,Z 357.954,A -85,B 0,C 180,E1 -24650.84,E2 -24650.84} C_VEL
LIN {X 0,Y 136.779,Z 355.241,A -85,B 0,C 180,E1 -24656.318,E2 -24656.318} C_VEL
LIN {X 0,Y 137.109,Z 354.535,A -85,B 0,C 180,E1 -24660,E2 -24660} C_VEL
LIN {X 0,Y 136.706,Z 355.371,A -85,B 0,C 180,E1 -24665.717,E2 -24665.717} C_VEL
LIN {X 0,Y 139.895,Z 359.898,A -85,B 0,C 180,E1 -24675.293,E2 -24675.293} C_VEL
LIN {X 0,Y 141.67,Z 360.958,A -85,B 0,C 180,E1 -24678.063,E2 -24678.063} C_VEL
LIN {X 0,Y 143.387,Z 364.147,A -85,B 0,C 180,E1 -24680.643,E2 -24680.643} C_VEL
LIN {X 0,Y 146.296,Z 366.506,A -85,B 0,C 180,E1 -24683.914,E2 -24683.914} C_VEL
LIN {X 0,Y 148.292,Z 369.766,A -85,B 0,C 180,E1 -24686.042,E2 -24686.042} C_VEL
LIN {X 0,Y 150.467,Z 371.9,A -85,B 0,C 180,E1 -24687.981,E2 -24687.981} C_VEL
LIN {X 0,Y 153.034,Z 375.497,A -85,B 0,C 180,E1 -24690.153,E2 -24690.153} C_VEL
LIN {X 0,Y 154.343,Z 377.133,A -85,B 0,C 180,E1 -24691.161,E2 -24691.161} C_VEL
LIN {X 0,Y 157.676,Z 381.777,A -85,B 0,C 180,E1 -24693.572,E2 -24693.572} C_VEL
LIN {X 0,Y 162.206,Z 388.379,A -85,B 0,C 180,E1 -24696.493,E2 -24696.493} C_VEL
LIN {X 0,Y 168.598,Z 398.846,A -85,B 0,C 180,E1 -24700.132,E2 -24700.132} C_VEL
LIN {X 0,Y 173.967,Z 408.915,A -85,B 0,C 180,E1 -24702.871,E2 -24702.871} C_VEL
LIN {X 0,Y 176.039,Z 413.233,A -85,B 0,C 180,E1 -24703.873,E2 -24703.873} C_VEL
LIN {X 0,Y 174.626,Z 441.286,A -85,B 0,C 180,E1 -24705.139,E2 -24705.139} C_VEL
LIN {X 0,Y 173.115,Z 454.497,A -85,B 0,C 180,E1 -24706.135,E2 -24706.135} C_VEL
LIN {X 0,Y 170.9,Z 466.919,A -85,B 0,C 180,E1 -24707.493,E2 -24707.493} C_VEL
LIN {X 0,Y 167.811,Z 479.235,A -85,B 0,C 180,E1 -24709.322,E2 -24709.322} C_VEL
LIN {X 0,Y 164.332,Z 489.696,A -85,B 0,C 180,E1 -24711.284,E2 -24711.284} C_VEL
LIN {X 0,Y 160.862,Z 498.744,A -85,B 0,C 180,E1 -24713.469,E2 -24713.469} C_VEL
LIN {X 0,Y 157.326,Z 507.14,A -85,B 0,C 180,E1 -24716.056,E2 -24716.056} C_VEL
LIN {X 0,Y 153.62,Z 514.873,A -85,B 0,C 180,E1 -24719.025,E2 -24719.025} C_VEL
LIN {X 0,Y 149.572,Z 522.525,A -85,B 0,C 180,E1 -24722.81,E2 -24722.81} C_VEL
LIN {X 0,Y 145.653,Z 529.322,A -85,B 0,C 180,E1 -24727.294,E2 -24727.294} C_VEL
LIN {X 0,Y 142.742,Z 533.928,A -85,B 0,C 180,E1 -24731.336,E2 -24731.336} C_VEL
LIN {X 0,Y 140.229,Z 537.473,A -85,B 0,C 180,E1 -24735.488,E2 -24735.488} C_VEL
LIN {X 0,Y 138.968,Z 539.295,A -85,B 0,C 180,E1 -24738.329,E2 -24738.329} C_VEL
LIN {X 0,Y 138.258,Z 540.624,A -85,B 0,C 180,E1 -24741.229,E2 -24741.229} C_VEL
LIN {X 0,Y 137.313,Z 542.168,A -85,B 0,C 180,E1 -24747.066,E2 -24747.066} C_VEL
LIN {X 0,Y 137.193,Z 542.389,A -85,B 0,C 180,E1 -24750,E2 -24750} C_VEL
LIN {X 0,Y 137.312,Z 542.198,A -85,B 0,C 180,E1 -24752.934,E2 -24752.934} C_VEL
LIN {X 0,Y 138.25,Z 540.693,A -85,B 0,C 180,E1 -24758.772,E2 -24758.772} C_VEL
LIN {X 0,Y 138.95,Z 539.395,A -85,B 0,C 180,E1 -24761.672,E2 -24761.672} C_VEL
LIN {X 0,Y 141.093,Z 536.549,A -85,B 0,C 180,E1 -24765.9,E2 -24765.9} C_VEL
LIN {X 0,Y 143.707,Z 532.713,A -85,B 0,C 180,E1 -24770.019,E2 -24770.019} C_VEL
LIN {X 0,Y 146.738,Z 527.623,A -85,B 0,C 180,E1 -24774.172,E2 -24774.172} C_VEL
LIN {X 0,Y 150.941,Z 520.37,A -85,B 0,C 180,E1 -24778.505,E2 -24778.505} C_VEL
LIN {X 0,Y 155.11,Z 512.332,A -85,B 0,C 180,E1 -24782.166,E2 -24782.166} C_VEL
LIN {X 0,Y 158.844,Z 504.099,A -85,B 0,C 180,E1 -24785.112,E2 -24785.112} C_VEL
LIN {X 0,Y 162.456,Z 495.051,A -85,B 0,C 180,E1 -24787.666,E2 -24787.666} C_VEL
LIN {X 0,Y 166.356,Z 484.495,A -85,B 0,C 180,E1 -24789.892,E2 -24789.892} C_VEL
LIN {X 0,Y 169.712,Z 472.789,A -85,B 0,C 180,E1 -24791.853,E2 -24791.853} C_VEL
LIN {X 0,Y 172.313,Z 461.284,A -85,B 0,C 180,E1 -24793.291,E2 -24793.291} C_VEL
LIN {X 0,Y 174.103,Z 448.534,A -85,B 0,C 180,E1 -24794.511,E2 -24794.511} C_VEL
LIN {X 0,Y 175.124,Z 436.556,A -85,B 0,C 180,E1 -24795.267,E2 -24795.267} C_VEL
LIN {X 0,Y 176.166,Z 413.297,A -85,B 0,C 180,E1 -24796.291,E2 -24796.291} C_VEL
LIN {X 0,Y 170.831,Z 402.731,A -85,B 0,C 180,E1 -24798.934,E2 -24798.934} C_VEL
LIN {X 0,Y 165.222,Z 393.076,A -85,B 0,C 180,E1 -24801.979,E2 -24801.979} C_VEL
LIN {X 0,Y 159.349,Z 384.013,A -85,B 0,C 180,E1 -24805.591,E2 -24805.591} C_VEL
LIN {X 0,Y 156.054,Z 379.5,A -85,B 0,C 180,E1 -24807.86,E2 -24807.86} C_VEL
LIN {X 0,Y 153.417,Z 375.739,A -85,B 0,C 180,E1 -24809.879,E2 -24809.879} C_VEL
LIN {X 0,Y 150.778,Z 372.296,A -85,B 0,C 180,E1 -24812.082,E2 -24812.082} C_VEL
LIN {X 0,Y 150.04,Z 371.323,A -85,B 0,C 180,E1 -24812.744,E2 -24812.744} C_VEL
LIN {X 0,Y 147.463,Z 368.616,A -85,B 0,C 180,E1 -24815.165,E2 -24815.165} C_VEL
LIN {X 0,Y 146.175,Z 366.24,A -85,B 0,C 180,E1 -24816.631,E2 -24816.631} C_VEL
LIN {X 0,Y 143.574,Z 364.328,A -85,B 0,C 180,E1 -24819.578,E2 -24819.578} C_VEL
LIN {X 0,Y 141.853,Z 361.378,A -85,B 0,C 180,E1 -24822.148,E2 -24822.148} C_VEL
LIN {X 0,Y 141.101,Z 360.436,A -85,B 0,C 180,E1 -24823.357,E2 -24823.357} C_VEL
LIN {X 0,Y 138.288,Z 358.398,A -85,B 0,C 180,E1 -24828.828,E2 -24828.828} C_VEL
LIN {X 0,Y 136.795,Z 355.307,A -85,B 0,C 180,E1 -24836.133,E2 -24836.133} C_VEL
LIN {X 0,Y 137.143,Z 354.698,A -85,B 0,C 180,E1 -24840,E2 -24840} C_VEL
LIN {X 0,Y 136.915,Z 355.62,A -85,B 0,C 180,E1 -24843.495,E2 -24843.495} C_VEL
LIN {X 0,Y 139.879,Z 359.778,A -85,B 0,C 180,E1 -24852.698,E2 -24852.698} C_VEL
LIN {X 0,Y 141.63,Z 360.927,A -85,B 0,C 180,E1 -24855.561,E2 -24855.561} C_VEL
LIN {X 0,Y 143.615,Z 364.273,A -85,B 0,C 180,E1 -24858.547,E2 -24858.547} C_VEL
LIN {X 0,Y 148.124,Z 371.164,A -85,B 0,C 180,E1 -24863.784,E2 -24863.784} C_VEL
LIN {X 0,Y 152.46,Z 378.491,A -85,B 0,C 180,E1 -24867.822,E2 -24867.822} C_VEL
LIN {X 0,Y 156.309,Z 385.534,A -85,B 0,C 180,E1 -24870.901,E2 -24870.901} C_VEL
LIN {X 0,Y 159.446,Z 391.637,A -85,B 0,C 180,E1 -24873.154,E2 -24873.154} C_VEL
LIN {X 0,Y 162.354,Z 397.755,A -85,B 0,C 180,E1 -24875.094,E2 -24875.094} C_VEL
LIN {X 0,Y 166.16,Z 406.304,A -85,B 0,C 180,E1 -24877.446,E2 -24877.446} C_VEL
LIN {X 0,Y 170.577,Z 417.597,A -85,B 0,C 180,E1 -24879.997,E2 -24879.997} C_VEL
LIN {X 0,Y 171.054,Z 419.895,A -85,B 0,C 180,E1 -24880.324,E2 -24880.324} C_VEL
LIN {X 0,Y 172.326,Z 448.969,A -85,B 0,C 180,E1 -24882.556,E2 -24882.556} C_VEL
LIN {X 0,Y 172.678,Z 464.368,A -85,B 0,C 180,E1 -24883.58,E2 -24883.58} C_VEL
LIN {X 0,Y 171.363,Z 478.886,A -85,B 0,C 180,E1 -24884.224,E2 -24884.224} C_VEL
LIN {X 0,Y 169.303,Z 491.255,A -85,B 0,C 180,E1 -24885.115,E2 -24885.115} C_VEL
LIN {X 0,Y 166.279,Z 503.875,A -85,B 0,C 180,E1 -24886.413,E2 -24886.413} C_VEL
LIN {X 0,Y 162.747,Z 515.19,A -85,B 0,C 180,E1 -24887.984,E2 -24887.984} C_VEL
LIN {X 0,Y 158.683,Z 526.218,A -85,B 0,C 180,E1 -24890.045,E2 -24890.045} C_VEL
LIN {X 0,Y 153.762,Z 537.161,A -85,B 0,C 180,E1 -24892.728,E2 -24892.728} C_VEL
LIN {X 0,Y 149.396,Z 546.101,A -85,B 0,C 180,E1 -24895.632,E2 -24895.632} C_VEL
LIN {X 0,Y 144.825,Z 554.866,A -85,B 0,C 180,E1 -24899.368,E2 -24899.368} C_VEL
LIN {X 0,Y 141.081,Z 561.933,A -85,B 0,C 180,E1 -24903.363,E2 -24903.363} C_VEL
LIN {X 0,Y 138.054,Z 567.634,A -85,B 0,C 180,E1 -24907.555,E2 -24907.555} C_VEL
LIN {X 0,Y 136.109,Z 572.193,A -85,B 0,C 180,E1 -24911.953,E2 -24911.953} C_VEL
LIN {X 0,Y 135.05,Z 575.694,A -85,B 0,C 180,E1 -24916.457,E2 -24916.457} C_VEL
LIN {X 0,Y 134.848,Z 578.636,A -85,B 0,C 180,E1 -24921.989,E2 -24921.989} C_VEL
LIN {X 0,Y 135.587,Z 580.115,A -85,B 0,C 180,E1 -24927.029,E2 -24927.029} C_VEL
LIN {X 0,Y 136.255,Z 580.441,A -85,B 0,C 180,E1 -24930,E2 -24930} C_VEL
LIN {X 0,Y 135.252,Z 579.683,A -85,B 0,C 180,E1 -24934.616,E2 -24934.616} C_VEL
LIN {X 0,Y 134.805,Z 578.182,A -85,B 0,C 180,E1 -24938.998,E2 -24938.998} C_VEL
LIN {X 0,Y 135.042,Z 575.638,A -85,B 0,C 180,E1 -24943.544,E2 -24943.544} C_VEL
LIN {X 0,Y 135.826,Z 572.853,A -85,B 0,C 180,E1 -24947.205,E2 -24947.205} C_VEL
LIN {X 0,Y 136.014,Z 570.72,A -85,B 0,C 180,E1 -24949.525,E2 -24949.525} C_VEL
LIN {X 0,Y 135.084,Z 566.714,A -85,B 0,C 180,E1 -24953.343,E2 -24953.343} C_VEL
LIN {X 0,Y 134.705,Z 562.114,A -85,B 0,C 180,E1 -24957.068,E2 -24957.068} C_VEL
LIN {X 0,Y 135.726,Z 559.01,A -85,B 0,C 180,E1 -24959.152,E2 -24959.152} C_VEL
LIN {X 0,Y 140.267,Z 550.958,A -85,B 0,C 180,E1 -24963.445,E2 -24963.445} C_VEL
LIN {X 0,Y 144.436,Z 543.228,A -85,B 0,C 180,E1 -24966.588,E2 -24966.588} C_VEL
LIN {X 0,Y 149.188,Z 533.925,A -85,B 0,C 180,E1 -24969.491,E2 -24969.491} C_VEL
LIN {X 0,Y 153.853,Z 523.61,A -85,B 0,C 180,E1 -24971.917,E2 -24971.917} C_VEL
LIN {X 0,Y 158.102,Z 512.168,A -85,B 0,C 180,E1 -24973.992,E2 -24973.992} C_VEL
LIN {X 0,Y 161.762,Z 500.317,A -85,B 0,C 180,E1 -24975.573,E2 -24975.573} C_VEL
LIN {X 0,Y 164.747,Z 487.322,A -85,B 0,C 180,E1 -24976.815,E2 -24976.815} C_VEL
LIN {X 0,Y 166.688,Z 474.599,A -85,B 0,C 180,E1 -24977.648,E2 -24977.648} C_VEL
LIN {X 0,Y 167.586,Z 463.647,A -85,B 0,C 180,E1 -24978.134,E2 -24978.134} C_VEL
LIN {X 0,Y 166.734,Z 433.052,A -85,B 0,C 180,E1 -24980.395,E2 -24980.395} C_VEL
LIN {X 0,Y 166.131,Z 421.094,A -85,B 0,C 180,E1 -24981.426,E2 -24981.426} C_VEL
LIN {X 0,Y 161.631,Z 409.12,A -85,B 0,C 180,E1 -24984.261,E2 -24984.261} C_VEL
LIN {X 0,Y 157.22,Z 399.047,A -85,B 0,C 180,E1 -24987.275,E2 -24987.275} C_VEL
LIN {X 0,Y 154.3,Z 392.982,A -85,B 0,C 180,E1 -24989.46,E2 -24989.46} C_VEL
LIN {X 0,Y 151.719,Z 387.921,A -85,B 0,C 180,E1 -24991.56,E2 -24991.56} C_VEL
LIN {X 0,Y 148.8,Z 382.416,A -85,B 0,C 180,E1 -24994.188,E2 -24994.188} C_VEL
LIN {X 0,Y 144.892,Z 375.594,A -85,B 0,C 180,E1 -24998.271,E2 -24998.271} C_VEL
LIN {X 0,Y 141.256,Z 369.846,A -85,B 0,C 180,E1 -25003.004,E2 -25003.004} C_VEL
LIN {X 0,Y 140.003,Z 367.439,A -85,B 0,C 180,E1 -25005.092,E2 -25005.092} C_VEL
LIN {X 0,Y 136.84,Z 364.777,A -85,B 0,C 180,E1 -25011.509,E2 -25011.509} C_VEL
LIN {X 0,Y 135.582,Z 361.943,A -85,B 0,C 180,E1 -25017.401,E2 -25017.401} C_VEL
LIN {X 0,Y 135.397,Z 361.441,A -85,B 0,C 180,E1 -25020,E2 -25020} C_VEL
LIN {X 0,Y 135.689,Z 362.411,A -85,B 0,C 180,E1 -25025.573,E2 -25025.573} C_VEL
LIN {X 0,Y 138.656,Z 366.76,A -85,B 0,C 180,E1 -25034.681,E2 -25034.681} C_VEL
LIN {X 0,Y 140.182,Z 367.76,A -85,B 0,C 180,E1 -25037.224,E2 -25037.224} C_VEL
LIN {X 0,Y 142.131,Z 371.141,A -85,B 0,C 180,E1 -25040.251,E2 -25040.251} C_VEL
LIN {X 0,Y 144.525,Z 373.271,A -85,B 0,C 180,E1 -25043.083,E2 -25043.083} C_VEL
LIN {X 0,Y 146.755,Z 376.64,A -85,B 0,C 180,E1 -25045.531,E2 -25045.531} C_VEL
LIN {X 0,Y 148.417,Z 378.415,A -85,B 0,C 180,E1 -25047.093,E2 -25047.093} C_VEL
LIN {X 0,Y 151.257,Z 382.225,A -85,B 0,C 180,E1 -25049.583,E2 -25049.583} C_VEL
LIN {X 0,Y 155.18,Z 387.975,A -85,B 0,C 180,E1 -25052.639,E2 -25052.639} C_VEL
LIN {X 0,Y 159.299,Z 394.185,A -85,B 0,C 180,E1 -25055.455,E2 -25055.455} C_VEL
LIN {X 0,Y 165.128,Z 404.075,A -85,B 0,C 180,E1 -25058.991,E2 -25058.991} C_VEL
LIN {X 0,Y 170.069,Z 413.681,A -85,B 0,C 180,E1 -25061.688,E2 -25061.688} C_VEL
LIN {X 0,Y 171.157,Z 415.933,A -85,B 0,C 180,E1 -25062.25,E2 -25062.25} C_VEL
LIN {X 0,Y 169.729,Z 442.02,A -85,B 0,C 180,E1 -25063.444,E2 -25063.444} C_VEL
LIN {X 0,Y 168.086,Z 455.675,A -85,B 0,C 180,E1 -25064.49,E2 -25064.49} C_VEL
LIN {X 0,Y 165.786,Z 467.904,A -85,B 0,C 180,E1 -25065.851,E2 -25065.851} C_VEL
LIN {X 0,Y 162.832,Z 479.24,A -85,B 0,C 180,E1 -25067.536,E2 -25067.536} C_VEL
LIN {X 0,Y 159.371,Z 489.407,A -85,B 0,C 180,E1 -25069.425,E2 -25069.425} C_VEL
LIN {X 0,Y 155.673,Z 498.682,A -85,B 0,C 180,E1 -25071.63,E2 -25071.63} C_VEL
LIN {X 0,Y 151.545,Z 508.121,A -85,B 0,C 180,E1 -25074.572,E2 -25074.572} C_VEL
LIN {X 0,Y 147.638,Z 515.853,A -85,B 0,C 180,E1 -25077.621,E2 -25077.621} C_VEL
LIN {X 0,Y 143.356,Z 523.504,A -85,B 0,C 180,E1 -25081.526,E2 -25081.526} C_VEL
LIN {X 0,Y 139.196,Z 530.302,A -85,B 0,C 180,E1 -25086.177,E2 -25086.177} C_VEL
LIN {X 0,Y 136.103,Z 534.907,A -85,B 0,C 180,E1 -25090.389,E2 -25090.389} C_VEL
LIN {X 0,Y 133.434,Z 538.453,A -85,B 0,C 180,E1 -25094.731,E2 -25094.731} C_VEL
LIN {X 0,Y 132.09,Z 540.274,A -85,B 0,C 180,E1 -25097.712,E2 -25097.712} C_VEL
LIN {X 0,Y 131.315,Z 541.603,A -85,B 0,C 180,E1 -25100.761,E2 -25100.761} C_VEL
LIN {X 0,Y 130.294,Z 543.146,A -85,B 0,C 180,E1 -25106.908,E2 -25106.908} C_VEL
LIN {X 0,Y 130.165,Z 543.367,A -85,B 0,C 180,E1 -25110,E2 -25110} C_VEL
LIN {X 0,Y 130.294,Z 543.176,A -85,B 0,C 180,E1 -25113.092,E2 -25113.092} C_VEL
LIN {X 0,Y 131.306,Z 541.67,A -85,B 0,C 180,E1 -25119.24,E2 -25119.24} C_VEL
LIN {X 0,Y 132.071,Z 540.373,A -85,B 0,C 180,E1 -25122.289,E2 -25122.289} C_VEL
LIN {X 0,Y 134.347,Z 537.526,A -85,B 0,C 180,E1 -25126.721,E2 -25126.721} C_VEL
LIN {X 0,Y 137.124,Z 533.69,A -85,B 0,C 180,E1 -25131.024,E2 -25131.024} C_VEL
LIN {X 0,Y 140.356,Z 528.599,A -85,B 0,C 180,E1 -25135.347,E2 -25135.347} C_VEL
LIN {X 0,Y 144.804,Z 521.346,A -85,B 0,C 180,E1 -25139.833,E2 -25139.833} C_VEL
LIN {X 0,Y 149.207,Z 513.308,A -85,B 0,C 180,E1 -25143.604,E2 -25143.604} C_VEL
LIN {X 0,Y 153.147,Z 505.074,A -85,B 0,C 180,E1 -25146.625,E2 -25146.625} C_VEL
LIN {X 0,Y 156.957,Z 496.024,A -85,B 0,C 180,E1 -25149.232,E2 -25149.232} C_VEL
LIN {X 0,Y 161.029,Z 485.467,A -85,B 0,C 180,E1 -25151.496,E2 -25151.496} C_VEL
LIN {X 0,Y 164.492,Z 473.918,A -85,B 0,C 180,E1 -25153.465,E2 -25153.465} C_VEL
LIN {X 0,Y 167.211,Z 462.598,A -85,B 0,C 180,E1 -25154.897,E2 -25154.897} C_VEL
LIN {X 0,Y 169.054,Z 450.43,A -85,B 0,C 180,E1 -25156.108,E2 -25156.108} C_VEL
LIN {X 0,Y 170.263,Z 437.038,A -85,B 0,C 180,E1 -25156.978,E2 -25156.978} C_VEL
LIN {X 0,Y 171.318,Z 416.1,A -85,B 0,C 180,E1 -25157.9,E2 -25157.9} C_VEL
LIN {X 0,Y 165.993,Z 405.507,A -85,B 0,C 180,E1 -25160.769,E2 -25160.769} C_VEL
